KUKA KRL program: EPS_2_251525_MH1778938_A_20251113053654.src

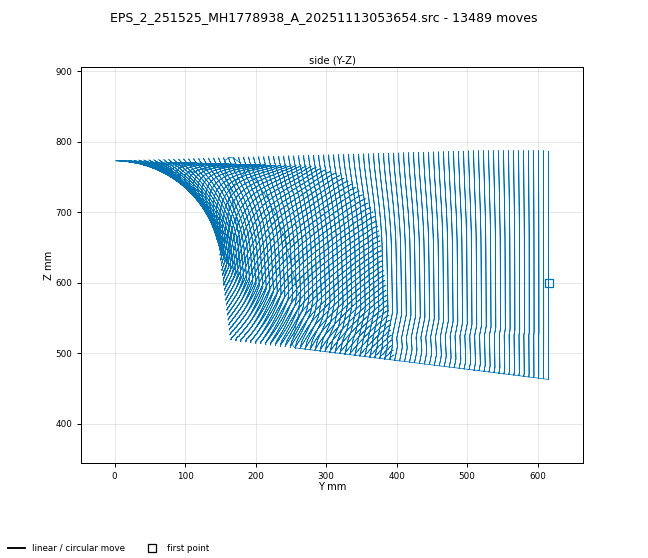
[picture p0: tool path of EPS_2_251525_MH1778938_A_20251113053654.src, 13489 of 13491 moves have a stored position in this frame; points joined in program order, loops and branches not executed]
&ACCESS RVP
&REL 4
&COMMENT QRS 19112012
&PARAM EDITMASK = *
DEF PART()
EXT BAS (BAS_COMMAND :IN,REAL :IN )
INT I
BAS (#INITMOV,0 )

;KUKA QRS Post kuka4.cps  Date:22-06-2017 !

File_ID=2903

QRS_PRE_INIT()

;Init var - Until changes are made in qrs_pre_init
Outlet_Square_prg=0
Inlet_1_Square_prg=0
Inlet_2_Square_prg=0
Inlet_3_Square_prg=0
Inlet_4_Square_prg=0
Inlet_5_Square_prg=0

Outlet_1={X 0.000, Y 516.340, Z 662.000, B 0.000, E1 0.000 }
Inlet_1={X 0.000, Y 535.290, Z 637.000, B 0.000, E1 180.000 }
Outlet_1_type=251
Inlet_1_type=0
;QRS#1=Sidecore dimensions
;QRS#2=250-10" PVC SDR 35
;QRS#3=DeadEnd 251
;QRS#4=
;QRS#5=
;QRS#6=
;QRS#7=
;QRS#8=
;QRS#9=14M PSX
;QRS#10=

;QRS#11=
;QRS#12=
;QRS#13=
;QRS#14=
;QRS#15=
;QRS#16=1220x127x1067 3,5'
;QRS#17=EPS Height
;QRS#18=787,5
;QRS#19=*
;QRS#20= UPDATED VERSION 22-06-2017
;QRS#21=*
Outlet_Square=0100
Inlet_1_Square=00
Inlet_2_Square=0
Inlet_3_Square=0
Inlet_4_Square=0
Inlet_5_Square=0
Mill_Square=1
Outlet_Square_Prg=205
Inlet_1_Square_prg=0

QRS_INIT()

$ADVANCE=5

; T1
PTP {E1 173.595,E2 173.595}
PTP {X 0,Y 615.507,A -85,B 0,C 180,E1 173.595,E2 173.595,E3 0,E4 0,E5 0,E6 0}
QRS_SPEED_INIT()
LIN {X 0,Y 615.507,Z 600,A -85,B 0,C 180,E1 173.595,E2 173.595,E3 0,E4 0,E5 0,E6 0} C_VEL
LIN {X 0,Y 615.507,Z 472.987,A -85,B 0,C 180,E1 173.595,E2 173.595} C_VEL
LIN {X 0,Y 615.507,Z 464.806,A -85,B 0,C 180,E1 173.595,E2 173.595} C_VEL
LIN {X 0,Y 615.49,Z 462.806,A -85,B 0,C 180,E1 173.409,E2 173.409} C_VEL
LIN {X 0,Y 615.478,Z 462.817,A -85,B 0,C 180,E1 170.801,E2 170.801} C_VEL
LIN {X 0,Y 615.479,Z 462.819,A -85,B 0,C 180,E1 168.139,E2 168.139} C_VEL
LIN {X 0,Y 615.488,Z 462.806,A -85,B 0,C 180,E1 165.451,E2 165.451} C_VEL
LIN {X 0,Y 615.479,Z 462.818,A -85,B 0,C 180,E1 162.73,E2 162.73} C_VEL
LIN {X 0,Y 615.477,Z 462.816,A -85,B 0,C 180,E1 159.967,E2 159.967} C_VEL
LIN {X 0,Y 615.482,Z 462.809,A -85,B 0,C 180,E1 157.156,E2 157.156} C_VEL
LIN {X 0,Y 615.494,Z 462.824,A -85,B 0,C 180,E1 154.285,E2 154.285} C_VEL
LIN {X 0,Y 615.486,Z 462.807,A -85,B 0,C 180,E1 151.342,E2 151.342} C_VEL
LIN {X 0,Y 615.477,Z 462.813,A -85,B 0,C 180,E1 148.913,E2 148.913} C_VEL
LIN {X 0,Y 615.485,Z 462.822,A -85,B 0,C 180,E1 146.464,E2 146.464} C_VEL
LIN {X 0,Y 615.481,Z 462.81,A -85,B 0,C 180,E1 143.575,E2 143.575} C_VEL
LIN {X 0,Y 615.479,Z 462.811,A -85,B 0,C 180,E1 140.937,E2 140.937} C_VEL
LIN {X 0,Y 615.482,Z 462.82,A -85,B 0,C 180,E1 138.526,E2 138.526} C_VEL
LIN {X 0,Y 615.478,Z 462.817,A -85,B 0,C 180,E1 135.85,E2 135.85} C_VEL
LIN {X 0,Y 615.485,Z 462.808,A -85,B 0,C 180,E1 133.048,E2 133.048} C_VEL
LIN {X 0,Y 615.49,Z 462.822,A -85,B 0,C 180,E1 130.09,E2 130.09} C_VEL
LIN {X 0,Y 615.49,Z 462.806,A -85,B 0,C 180,E1 127.241,E2 127.241} C_VEL
LIN {X 0,Y 615.476,Z 462.814,A -85,B 0,C 180,E1 124.7,E2 124.7} C_VEL
LIN {X 0,Y 615.488,Z 462.822,A -85,B 0,C 180,E1 122.332,E2 122.332} C_VEL
LIN {X 0,Y 615.478,Z 462.81,A -85,B 0,C 180,E1 119.406,E2 119.406} C_VEL
LIN {X 0,Y 615.491,Z 462.806,A -85,B 0,C 180,E1 117.047,E2 117.047} C_VEL
LIN {X 0,Y 615.487,Z 462.823,A -85,B 0,C 180,E1 114.271,E2 114.271} C_VEL
LIN {X 0,Y 615.48,Z 462.81,A -85,B 0,C 180,E1 111.432,E2 111.432} C_VEL
LIN {X 0,Y 615.477,Z 462.813,A -85,B 0,C 180,E1 108.646,E2 108.646} C_VEL
LIN {X 0,Y 615.486,Z 462.821,A -85,B 0,C 180,E1 105.905,E2 105.905} C_VEL
LIN {X 0,Y 615.487,Z 462.807,A -85,B 0,C 180,E1 103.201,E2 103.201} C_VEL
LIN {X 0,Y 615.476,Z 462.815,A -85,B 0,C 180,E1 100.527,E2 100.527} C_VEL
LIN {X 0,Y 615.487,Z 462.822,A -85,B 0,C 180,E1 97.875,E2 97.875} C_VEL
LIN {X 0,Y 615.479,Z 462.809,A -85,B 0,C 180,E1 95.241,E2 95.241} C_VEL
LIN {X 0,Y 615.478,Z 462.812,A -85,B 0,C 180,E1 92.618,E2 92.618} C_VEL
LIN {X 0,Y 615.486,Z 462.828,A -85,B 0,C 180,E1 90,E2 90} C_VEL
LIN {X 0,Y 615.478,Z 462.812,A -85,B 0,C 180,E1 87.382,E2 87.382} C_VEL
LIN {X 0,Y 615.483,Z 462.808,A -85,B 0,C 180,E1 84.759,E2 84.759} C_VEL
LIN {X 0,Y 615.487,Z 462.822,A -85,B 0,C 180,E1 82.125,E2 82.125} C_VEL
LIN {X 0,Y 615.476,Z 462.815,A -85,B 0,C 180,E1 79.473,E2 79.473} C_VEL
LIN {X 0,Y 615.487,Z 462.807,A -85,B 0,C 180,E1 76.799,E2 76.799} C_VEL
LIN {X 0,Y 615.486,Z 462.821,A -85,B 0,C 180,E1 74.095,E2 74.095} C_VEL
LIN {X 0,Y 615.477,Z 462.813,A -85,B 0,C 180,E1 71.354,E2 71.354} C_VEL
LIN {X 0,Y 615.48,Z 462.81,A -85,B 0,C 180,E1 68.568,E2 68.568} C_VEL
LIN {X 0,Y 615.487,Z 462.823,A -85,B 0,C 180,E1 65.729,E2 65.729} C_VEL
LIN {X 0,Y 615.487,Z 462.807,A -85,B 0,C 180,E1 62.824,E2 62.824} C_VEL
LIN {X 0,Y 615.499,Z 462.825,A -85,B 0,C 180,E1 59.841,E2 59.841} C_VEL
LIN {X 0,Y 615.481,Z 462.819,A -85,B 0,C 180,E1 57.543,E2 57.543} C_VEL
LIN {X 0,Y 615.478,Z 462.812,A -85,B 0,C 180,E1 55.185,E2 55.185} C_VEL
LIN {X 0,Y 615.491,Z 462.806,A -85,B 0,C 180,E1 52.759,E2 52.759} C_VEL
LIN {X 0,Y 615.49,Z 462.822,A -85,B 0,C 180,E1 49.91,E2 49.91} C_VEL
LIN {X 0,Y 615.485,Z 462.808,A -85,B 0,C 180,E1 46.952,E2 46.952} C_VEL
LIN {X 0,Y 615.482,Z 462.82,A -85,B 0,C 180,E1 43.998,E2 43.998} C_VEL
LIN {X 0,Y 615.478,Z 462.811,A -85,B 0,C 180,E1 41.095,E2 41.095} C_VEL
LIN {X 0,Y 615.484,Z 462.808,A -85,B 0,C 180,E1 38.904,E2 38.904} C_VEL
LIN {X 0,Y 615.481,Z 462.81,A -85,B 0,C 180,E1 36.425,E2 36.425} C_VEL
LIN {X 0,Y 615.485,Z 462.822,A -85,B 0,C 180,E1 33.536,E2 33.536} C_VEL
LIN {X 0,Y 615.482,Z 462.809,A -85,B 0,C 180,E1 30.919,E2 30.919} C_VEL
LIN {X 0,Y 615.483,Z 462.808,A -85,B 0,C 180,E1 28.452,E2 28.452} C_VEL
LIN {X 0,Y 615.493,Z 462.824,A -85,B 0,C 180,E1 25.573,E2 25.573} C_VEL
LIN {X 0,Y 615.482,Z 462.809,A -85,B 0,C 180,E1 22.844,E2 22.844} C_VEL
LIN {X 0,Y 615.477,Z 462.816,A -85,B 0,C 180,E1 20.033,E2 20.033} C_VEL
LIN {X 0,Y 615.479,Z 462.818,A -85,B 0,C 180,E1 17.27,E2 17.27} C_VEL
LIN {X 0,Y 615.488,Z 462.806,A -85,B 0,C 180,E1 14.549,E2 14.549} C_VEL
LIN {X 0,Y 615.479,Z 462.819,A -85,B 0,C 180,E1 11.861,E2 11.861} C_VEL
LIN {X 0,Y 615.478,Z 462.817,A -85,B 0,C 180,E1 9.199,E2 9.199} C_VEL
LIN {X 0,Y 615.491,Z 462.806,A -85,B 0,C 180,E1 6.556,E2 6.556} C_VEL
LIN {X 0,Y 615.478,Z 462.817,A -85,B 0,C 180,E1 3.928,E2 3.928} C_VEL
LIN {X 0,Y 615.485,Z 462.821,A -85,B 0,C 180,E1 1.308,E2 1.308} C_VEL
LIN {X 0,Y 615.485,Z 462.808,A -85,B 0,C 180,E1 -1.309,E2 -1.309} C_VEL
LIN {X 0,Y 615.478,Z 462.812,A -85,B 0,C 180,E1 -3.929,E2 -3.929} C_VEL
LIN {X 0,Y 615.489,Z 462.825,A -85,B 0,C 180,E1 -6.591,E2 -6.591} C_VEL
LIN {X 0,Y 615.478,Z 462.811,A -85,B 0,C 180,E1 -9.199,E2 -9.199} C_VEL
LIN {X 0,Y 615.481,Z 462.81,A -85,B 0,C 180,E1 -11.861,E2 -11.861} C_VEL
LIN {X 0,Y 615.488,Z 462.827,A -85,B 0,C 180,E1 -14.549,E2 -14.549} C_VEL
LIN {X 0,Y 615.478,Z 462.811,A -85,B 0,C 180,E1 -17.271,E2 -17.271} C_VEL
LIN {X 0,Y 615.477,Z 462.813,A -85,B 0,C 180,E1 -20.033,E2 -20.033} C_VEL
LIN {X 0,Y 615.482,Z 462.821,A -85,B 0,C 180,E1 -22.845,E2 -22.845} C_VEL
LIN {X 0,Y 615.493,Z 462.805,A -85,B 0,C 180,E1 -25.716,E2 -25.716} C_VEL
LIN {X 0,Y 615.486,Z 462.828,A -85,B 0,C 180,E1 -28.658,E2 -28.658} C_VEL
LIN {X 0,Y 615.477,Z 462.816,A -85,B 0,C 180,E1 -31.087,E2 -31.087} C_VEL
LIN {X 0,Y 615.485,Z 462.808,A -85,B 0,C 180,E1 -33.536,E2 -33.536} C_VEL
LIN {X 0,Y 615.482,Z 462.819,A -85,B 0,C 180,E1 -36.425,E2 -36.425} C_VEL
LIN {X 0,Y 615.478,Z 462.818,A -85,B 0,C 180,E1 -39.063,E2 -39.063} C_VEL
LIN {X 0,Y 615.482,Z 462.809,A -85,B 0,C 180,E1 -41.475,E2 -41.475} C_VEL
LIN {X 0,Y 615.478,Z 462.812,A -85,B 0,C 180,E1 -44.151,E2 -44.151} C_VEL
LIN {X 0,Y 615.485,Z 462.821,A -85,B 0,C 180,E1 -46.953,E2 -46.953} C_VEL
LIN {X 0,Y 615.478,Z 462.812,A -85,B 0,C 180,E1 -49.394,E2 -49.394} C_VEL
LIN {X 0,Y 615.485,Z 462.808,A -85,B 0,C 180,E1 -51.989,E2 -51.989} C_VEL
LIN {X 0,Y 615.474,Z 462.817,A -85,B 0,C 180,E1 -54.384,E2 -54.384} C_VEL
LIN {X 0,Y 615.484,Z 462.827,A -85,B 0,C 180,E1 -56.764,E2 -56.764} C_VEL
LIN {X 0,Y 615.478,Z 462.82,A -85,B 0,C 180,E1 -59.081,E2 -59.081} C_VEL
LIN {X 0,Y 615.48,Z 462.81,A -85,B 0,C 180,E1 -61.551,E2 -61.551} C_VEL
LIN {X 0,Y 615.477,Z 462.813,A -85,B 0,C 180,E1 -64.284,E2 -64.284} C_VEL
LIN {X 0,Y 615.497,Z 463.131,A -85,B 0,C 180,E1 -64.973,E2 -64.973} C_VEL
LIN {X 0,Y 615.483,Z 480.491,A -85,B 0,C 180,E1 -67.655,E2 -67.655} C_VEL
LIN {X 0,Y 615.475,Z 498.123,A -85,B 0,C 180,E1 -70.315,E2 -70.315} C_VEL
LIN {X 0,Y 615.495,Z 516.688,A -85,B 0,C 180,E1 -73.072,E2 -73.072} C_VEL
LIN {X 0,Y 615.49,Z 525.925,A -85,B 0,C 180,E1 -74.393,E2 -74.393} C_VEL
LIN {X 0,Y 615.49,Z 528.646,A -85,B 0,C 180,E1 -74.456,E2 -74.456} C_VEL
LIN {X 0,Y 615.499,Z 662.918,A -85,B 0,C 180,E1 -76.064,E2 -76.064} C_VEL
LIN {X 0,Y 615.497,Z 677.388,A -85,B 0,C 180,E1 -76.379,E2 -76.379} C_VEL
LIN {X 0,Y 615.498,Z 690.696,A -85,B 0,C 180,E1 -76.799,E2 -76.799} C_VEL
LIN {X 0,Y 615.495,Z 702.843,A -85,B 0,C 180,E1 -77.303,E2 -77.303} C_VEL
LIN {X 0,Y 615.492,Z 715.604,A -85,B 0,C 180,E1 -77.972,E2 -77.972} C_VEL
LIN {X 0,Y 615.499,Z 728.344,A -85,B 0,C 180,E1 -78.807,E2 -78.807} C_VEL
LIN {X 0,Y 615.498,Z 738.751,A -85,B 0,C 180,E1 -79.64,E2 -79.64} C_VEL
LIN {X 0,Y 615.497,Z 749.09,A -85,B 0,C 180,E1 -80.636,E2 -80.636} C_VEL
LIN {X 0,Y 615.497,Z 757.604,A -85,B 0,C 180,E1 -81.629,E2 -81.629} C_VEL
LIN {X 0,Y 615.496,Z 765.727,A -85,B 0,C 180,E1 -82.785,E2 -82.785} C_VEL
LIN {X 0,Y 615.497,Z 771.431,A -85,B 0,C 180,E1 -83.773,E2 -83.773} C_VEL
LIN {X 0,Y 615.495,Z 776.081,A -85,B 0,C 180,E1 -84.759,E2 -84.759} C_VEL
LIN {X 0,Y 615.494,Z 780.902,A -85,B 0,C 180,E1 -86.072,E2 -86.072} C_VEL
LIN {X 0,Y 615.496,Z 784.252,A -85,B 0,C 180,E1 -87.382,E2 -87.382} C_VEL
LIN {X 0,Y 615.489,Z 786.229,A -85,B 0,C 180,E1 -88.691,E2 -88.691} C_VEL
LIN {X 0,Y 615.493,Z 786.889,A -85,B 0,C 180,E1 -90,E2 -90} C_VEL
LIN {X 0,Y 615.489,Z 786.229,A -85,B 0,C 180,E1 -91.309,E2 -91.309} C_VEL
LIN {X 0,Y 615.496,Z 784.252,A -85,B 0,C 180,E1 -92.618,E2 -92.618} C_VEL
LIN {X 0,Y 615.494,Z 780.902,A -85,B 0,C 180,E1 -93.928,E2 -93.928} C_VEL
LIN {X 0,Y 615.495,Z 776.081,A -85,B 0,C 180,E1 -95.241,E2 -95.241} C_VEL
LIN {X 0,Y 615.495,Z 769.629,A -85,B 0,C 180,E1 -96.556,E2 -96.556} C_VEL
LIN {X 0,Y 615.497,Z 762.442,A -85,B 0,C 180,E1 -97.71,E2 -97.71} C_VEL
LIN {X 0,Y 615.497,Z 754.905,A -85,B 0,C 180,E1 -98.702,E2 -98.702} C_VEL
LIN {X 0,Y 615.495,Z 745.855,A -85,B 0,C 180,E1 -99.696,E2 -99.696} C_VEL
LIN {X 0,Y 615.497,Z 735.759,A -85,B 0,C 180,E1 -100.618,E2 -100.618} C_VEL
LIN {X 0,Y 615.498,Z 724.861,A -85,B 0,C 180,E1 -101.443,E2 -101.443} C_VEL
LIN {X 0,Y 615.487,Z 712.711,A -85,B 0,C 180,E1 -102.195,E2 -102.195} C_VEL
LIN {X 0,Y 615.494,Z 699.097,A -85,B 0,C 180,E1 -102.865,E2 -102.865} C_VEL
LIN {X 0,Y 615.497,Z 685.843,A -85,B 0,C 180,E1 -103.369,E2 -103.369} C_VEL
LIN {X 0,Y 615.498,Z 672.298,A -85,B 0,C 180,E1 -103.747,E2 -103.747} C_VEL
LIN {X 0,Y 615.497,Z 657.754,A -85,B 0,C 180,E1 -104.013,E2 -104.013} C_VEL
LIN {X 0,Y 615.49,Z 526.279,A -85,B 0,C 180,E1 -105.586,E2 -105.586} C_VEL
LIN {X 0,Y 615.49,Z 524.805,A -85,B 0,C 180,E1 -105.735,E2 -105.735} C_VEL
LIN {X 0,Y 615.479,Z 506.472,A -85,B 0,C 180,E1 -108.44,E2 -108.44} C_VEL
LIN {X 0,Y 615.497,Z 487.671,A -85,B 0,C 180,E1 -111.255,E2 -111.255} C_VEL
LIN {X 0,Y 615.497,Z 469.607,A -85,B 0,C 180,E1 -114.01,E2 -114.01} C_VEL
LIN {X 0,Y 615.497,Z 463,A -85,B 0,C 180,E1 -115.062,E2 -115.062} C_VEL
LIN {X 0,Y 615.487,Z 462.828,A -85,B 0,C 180,E1 -117.177,E2 -117.177} C_VEL
LIN {X 0,Y 615.499,Z 462.804,A -85,B 0,C 180,E1 -120.159,E2 -120.159} C_VEL
LIN {X 0,Y 615.481,Z 462.81,A -85,B 0,C 180,E1 -122.457,E2 -122.457} C_VEL
LIN {X 0,Y 615.477,Z 462.817,A -85,B 0,C 180,E1 -124.815,E2 -124.815} C_VEL
LIN {X 0,Y 615.491,Z 462.826,A -85,B 0,C 180,E1 -127.241,E2 -127.241} C_VEL
LIN {X 0,Y 615.489,Z 462.807,A -85,B 0,C 180,E1 -130.089,E2 -130.089} C_VEL
LIN {X 0,Y 615.49,Z 462.806,A -85,B 0,C 180,E1 -132.352,E2 -132.352} C_VEL
LIN {X 0,Y 615.479,Z 462.822,A -85,B 0,C 180,E1 -135.068,E2 -135.068} C_VEL
LIN {X 0,Y 615.477,Z 462.812,A -85,B 0,C 180,E1 -137.919,E2 -137.919} C_VEL
LIN {X 0,Y 615.498,Z 462.804,A -85,B 0,C 180,E1 -140.25,E2 -140.25} C_VEL
LIN {X 0,Y 615.478,Z 462.821,A -85,B 0,C 180,E1 -143.063,E2 -143.063} C_VEL
LIN {X 0,Y 615.49,Z 462.827,A -85,B 0,C 180,E1 -145.297,E2 -145.297} C_VEL
LIN {X 0,Y 615.479,Z 462.818,A -85,B 0,C 180,E1 -147.668,E2 -147.668} C_VEL
LIN {X 0,Y 615.488,Z 462.807,A -85,B 0,C 180,E1 -150.203,E2 -150.203} C_VEL
LIN {X 0,Y 615.477,Z 462.817,A -85,B 0,C 180,E1 -152.954,E2 -152.954} C_VEL
LIN {X 0,Y 615.479,Z 462.818,A -85,B 0,C 180,E1 -155.727,E2 -155.727} C_VEL
LIN {X 0,Y 615.486,Z 462.808,A -85,B 0,C 180,E1 -158.568,E2 -158.568} C_VEL
LIN {X 0,Y 615.492,Z 462.826,A -85,B 0,C 180,E1 -161.39,E2 -161.39} C_VEL
LIN {X 0,Y 615.48,Z 462.811,A -85,B 0,C 180,E1 -164.094,E2 -164.094} C_VEL
LIN {X 0,Y 615.478,Z 462.812,A -85,B 0,C 180,E1 -166.798,E2 -166.798} C_VEL
LIN {X 0,Y 615.489,Z 462.827,A -85,B 0,C 180,E1 -169.473,E2 -169.473} C_VEL
LIN {X 0,Y 615.479,Z 462.811,A -85,B 0,C 180,E1 -172.124,E2 -172.124} C_VEL
LIN {X 0,Y 615.481,Z 462.81,A -85,B 0,C 180,E1 -174.758,E2 -174.758} C_VEL
LIN {X 0,Y 615.491,Z 462.823,A -85,B 0,C 180,E1 -177.382,E2 -177.382} C_VEL
LIN {X 0,Y 615.477,Z 462.815,A -85,B 0,C 180,E1 -180,E2 -180} C_VEL
LIN {X 0,Y 615.491,Z 462.806,A -85,B 0,C 180,E1 -182.618,E2 -182.618} C_VEL
LIN {X 0,Y 615.476,Z 462.82,A -85,B 0,C 180,E1 -185.241,E2 -185.241} C_VEL
LIN {X 0,Y 615.49,Z 462.806,A -85,B 0,C 180,E1 -186.591,E2 -186.591} C_VEL
LIN {X 0,Y 614.807,Z 462.965,A -85,B 0,C 180,E1 -187.137,E2 -187.137} C_VEL
LIN {X 0,Y 611.966,Z 463.377,A -85,B 0,C 180,E1 -188.023,E2 -188.023} C_VEL
LIN {X 0,Y 609.574,Z 463.69,A -85,B 0,C 180,E1 -188.736,E2 -188.736} C_VEL
LIN {X 0,Y 608.539,Z 463.808,A -85,B 0,C 180,E1 -189.286,E2 -189.286} C_VEL
LIN {X 0,Y 608.451,Z 463.817,A -85,B 0,C 180,E1 -189.472,E2 -189.472} C_VEL
LIN {X 0,Y 608.456,Z 463.815,A -85,B 0,C 180,E1 -192,E2 -192} C_VEL
LIN {X 0,Y 608.472,Z 463.81,A -85,B 0,C 180,E1 -194.72,E2 -194.72} C_VEL
LIN {X 0,Y 608.445,Z 463.821,A -85,B 0,C 180,E1 -197.476,E2 -197.476} C_VEL
LIN {X 0,Y 608.458,Z 463.813,A -85,B 0,C 180,E1 -200.274,E2 -200.274} C_VEL
LIN {X 0,Y 608.449,Z 463.812,A -85,B 0,C 180,E1 -202.477,E2 -202.477} C_VEL
LIN {X 0,Y 608.45,Z 463.817,A -85,B 0,C 180,E1 -205.301,E2 -205.301} C_VEL
LIN {X 0,Y 608.442,Z 463.822,A -85,B 0,C 180,E1 -207.518,E2 -207.518} C_VEL
LIN {X 0,Y 608.464,Z 463.816,A -85,B 0,C 180,E1 -209.973,E2 -209.973} C_VEL
LIN {X 0,Y 608.457,Z 463.812,A -85,B 0,C 180,E1 -212.524,E2 -212.524} C_VEL
LIN {X 0,Y 608.449,Z 463.816,A -85,B 0,C 180,E1 -215.277,E2 -215.277} C_VEL
LIN {X 0,Y 608.46,Z 463.814,A -85,B 0,C 180,E1 -218.241,E2 -218.241} C_VEL
LIN {X 0,Y 608.446,Z 463.814,A -85,B 0,C 180,E1 -220.33,E2 -220.33} C_VEL
LIN {X 0,Y 608.446,Z 463.813,A -85,B 0,C 180,E1 -222.96,E2 -222.96} C_VEL
LIN {X 0,Y 608.459,Z 463.822,A -85,B 0,C 180,E1 -225.735,E2 -225.735} C_VEL
LIN {X 0,Y 608.459,Z 463.811,A -85,B 0,C 180,E1 -228.657,E2 -228.657} C_VEL
LIN {X 0,Y 608.465,Z 463.815,A -85,B 0,C 180,E1 -231.413,E2 -231.413} C_VEL
LIN {X 0,Y 608.47,Z 463.818,A -85,B 0,C 180,E1 -233.951,E2 -233.951} C_VEL
LIN {X 0,Y 608.459,Z 463.814,A -85,B 0,C 180,E1 -236.33,E2 -236.33} C_VEL
LIN {X 0,Y 608.473,Z 463.81,A -85,B 0,C 180,E1 -238.727,E2 -238.727} C_VEL
LIN {X 0,Y 608.466,Z 463.814,A -85,B 0,C 180,E1 -241.38,E2 -241.38} C_VEL
LIN {X 0,Y 608.439,Z 463.823,A -85,B 0,C 180,E1 -243.965,E2 -243.965} C_VEL
LIN {X 0,Y 608.466,Z 463.816,A -85,B 0,C 180,E1 -246.156,E2 -246.156} C_VEL
LIN {X 0,Y 608.467,Z 463.814,A -85,B 0,C 180,E1 -248.309,E2 -248.309} C_VEL
LIN {X 0,Y 608.45,Z 463.813,A -85,B 0,C 180,E1 -251.131,E2 -251.131} C_VEL
LIN {X 0,Y 608.458,Z 463.823,A -85,B 0,C 180,E1 -253.907,E2 -253.907} C_VEL
LIN {X 0,Y 608.464,Z 463.811,A -85,B 0,C 180,E1 -256.644,E2 -256.644} C_VEL
LIN {X 0,Y 608.458,Z 463.813,A -85,B 0,C 180,E1 -259.35,E2 -259.35} C_VEL
LIN {X 0,Y 608.476,Z 463.819,A -85,B 0,C 180,E1 -262.033,E2 -262.033} C_VEL
LIN {X 0,Y 608.46,Z 463.812,A -85,B 0,C 180,E1 -264.698,E2 -264.698} C_VEL
LIN {X 0,Y 608.469,Z 463.811,A -85,B 0,C 180,E1 -267.352,E2 -267.352} C_VEL
LIN {X 0,Y 608.476,Z 463.82,A -85,B 0,C 180,E1 -270,E2 -270} C_VEL
LIN {X 0,Y 608.469,Z 463.811,A -85,B 0,C 180,E1 -272.648,E2 -272.648} C_VEL
LIN {X 0,Y 608.463,Z 463.812,A -85,B 0,C 180,E1 -275.302,E2 -275.302} C_VEL
LIN {X 0,Y 608.476,Z 463.819,A -85,B 0,C 180,E1 -277.967,E2 -277.967} C_VEL
LIN {X 0,Y 608.458,Z 463.813,A -85,B 0,C 180,E1 -280.65,E2 -280.65} C_VEL
LIN {X 0,Y 608.464,Z 463.811,A -85,B 0,C 180,E1 -283.356,E2 -283.356} C_VEL
LIN {X 0,Y 608.458,Z 463.823,A -85,B 0,C 180,E1 -286.093,E2 -286.093} C_VEL
LIN {X 0,Y 608.45,Z 463.813,A -85,B 0,C 180,E1 -288.869,E2 -288.869} C_VEL
LIN {X 0,Y 608.467,Z 463.814,A -85,B 0,C 180,E1 -291.691,E2 -291.691} C_VEL
LIN {X 0,Y 608.454,Z 463.815,A -85,B 0,C 180,E1 -294.57,E2 -294.57} C_VEL
LIN {X 0,Y 608.48,Z 463.809,A -85,B 0,C 180,E1 -297.209,E2 -297.209} C_VEL
LIN {X 0,Y 608.466,Z 463.818,A -85,B 0,C 180,E1 -299.972,E2 -299.972} C_VEL
LIN {X 0,Y 608.456,Z 463.816,A -85,B 0,C 180,E1 -302.522,E2 -302.522} C_VEL
LIN {X 0,Y 608.433,Z 463.814,A -85,B 0,C 180,E1 -305.277,E2 -305.277} C_VEL
LIN {X 0,Y 608.47,Z 463.813,A -85,B 0,C 180,E1 -307.745,E2 -307.745} C_VEL
LIN {X 0,Y 608.474,Z 463.818,A -85,B 0,C 180,E1 -310.332,E2 -310.332} C_VEL
LIN {X 0,Y 608.484,Z 463.807,A -85,B 0,C 180,E1 -313.311,E2 -313.311} C_VEL
LIN {X 0,Y 608.466,Z 463.819,A -85,B 0,C 180,E1 -316.131,E2 -316.131} C_VEL
LIN {X 0,Y 608.448,Z 463.814,A -85,B 0,C 180,E1 -318.823,E2 -318.823} C_VEL
LIN {X 0,Y 608.464,Z 463.811,A -85,B 0,C 180,E1 -321.412,E2 -321.412} C_VEL
LIN {X 0,Y 608.47,Z 463.815,A -85,B 0,C 180,E1 -323.95,E2 -323.95} C_VEL
LIN {X 0,Y 608.461,Z 463.822,A -85,B 0,C 180,E1 -326.33,E2 -326.33} C_VEL
LIN {X 0,Y 608.468,Z 463.814,A -85,B 0,C 180,E1 -328.727,E2 -328.727} C_VEL
LIN {X 0,Y 608.471,Z 463.81,A -85,B 0,C 180,E1 -331.378,E2 -331.378} C_VEL
LIN {X 0,Y 608.475,Z 463.819,A -85,B 0,C 180,E1 -334.276,E2 -334.276} C_VEL
LIN {X 0,Y 608.447,Z 463.815,A -85,B 0,C 180,E1 -336.876,E2 -336.876} C_VEL
LIN {X 0,Y 608.464,Z 463.81,A -85,B 0,C 180,E1 -339.319,E2 -339.319} C_VEL
LIN {X 0,Y 608.446,Z 463.815,A -85,B 0,C 180,E1 -341.828,E2 -341.828} C_VEL
LIN {X 0,Y 608.463,Z 463.818,A -85,B 0,C 180,E1 -344.594,E2 -344.594} C_VEL
LIN {X 0,Y 608.475,Z 463.809,A -85,B 0,C 180,E1 -347.323,E2 -347.323} C_VEL
LIN {X 0,Y 608.45,Z 463.816,A -85,B 0,C 180,E1 -350.023,E2 -350.023} C_VEL
LIN {X 0,Y 608.474,Z 463.816,A -85,B 0,C 180,E1 -352.701,E2 -352.701} C_VEL
LIN {X 0,Y 608.463,Z 463.811,A -85,B 0,C 180,E1 -355.363,E2 -355.363} C_VEL
LIN {X 0,Y 608.448,Z 463.815,A -85,B 0,C 180,E1 -358.015,E2 -358.015} C_VEL
LIN {X 0,Y 608.478,Z 463.817,A -85,B 0,C 180,E1 -360.662,E2 -360.662} C_VEL
LIN {X 0,Y 608.475,Z 463.809,A -85,B 0,C 180,E1 -363.311,E2 -363.311} C_VEL
LIN {X 0,Y 608.453,Z 463.814,A -85,B 0,C 180,E1 -365.967,E2 -365.967} C_VEL
LIN {X 0,Y 608.456,Z 463.821,A -85,B 0,C 180,E1 -368.636,E2 -368.636} C_VEL
LIN {X 0,Y 608.468,Z 463.81,A -85,B 0,C 180,E1 -371.324,E2 -371.324} C_VEL
LIN {X 0,Y 608.458,Z 463.813,A -85,B 0,C 180,E1 -374.038,E2 -374.038} C_VEL
LIN {X 0,Y 608.472,Z 463.817,A -85,B 0,C 180,E1 -376.784,E2 -376.784} C_VEL
LIN {X 0,Y 608.445,Z 463.813,A -85,B 0,C 180,E1 -379.571,E2 -379.571} C_VEL
LIN {X 0,Y 608.467,Z 463.817,A -85,B 0,C 180,E1 -382.406,E2 -382.406} C_VEL
LIN {X 0,Y 608.446,Z 463.823,A -85,B 0,C 180,E1 -384.572,E2 -384.572} C_VEL
LIN {X 0,Y 608.47,Z 463.812,A -85,B 0,C 180,E1 -387.208,E2 -387.208} C_VEL
LIN {X 0,Y 608.464,Z 463.812,A -85,B 0,C 180,E1 -389.973,E2 -389.973} C_VEL
LIN {X 0,Y 608.458,Z 463.82,A -85,B 0,C 180,E1 -392.524,E2 -392.524} C_VEL
LIN {X 0,Y 608.449,Z 463.814,A -85,B 0,C 180,E1 -395.278,E2 -395.278} C_VEL
LIN {X 0,Y 608.461,Z 463.814,A -85,B 0,C 180,E1 -398.241,E2 -398.241} C_VEL
LIN {X 0,Y 608.446,Z 463.817,A -85,B 0,C 180,E1 -400.33,E2 -400.33} C_VEL
LIN {X 0,Y 608.445,Z 463.82,A -85,B 0,C 180,E1 -402.961,E2 -402.961} C_VEL
LIN {X 0,Y 608.459,Z 463.811,A -85,B 0,C 180,E1 -405.736,E2 -405.736} C_VEL
LIN {X 0,Y 608.46,Z 463.82,A -85,B 0,C 180,E1 -408.658,E2 -408.658} C_VEL
LIN {X 0,Y 608.465,Z 463.811,A -85,B 0,C 180,E1 -411.413,E2 -411.413} C_VEL
LIN {X 0,Y 608.443,Z 463.812,A -85,B 0,C 180,E1 -413.955,E2 -413.955} C_VEL
LIN {X 0,Y 608.463,Z 463.814,A -85,B 0,C 180,E1 -416.33,E2 -416.33} C_VEL
LIN {X 0,Y 608.476,Z 463.819,A -85,B 0,C 180,E1 -418.728,E2 -418.728} C_VEL
LIN {X 0,Y 608.466,Z 463.812,A -85,B 0,C 180,E1 -421.382,E2 -421.382} C_VEL
LIN {X 0,Y 608.438,Z 463.815,A -85,B 0,C 180,E1 -423.965,E2 -423.965} C_VEL
LIN {X 0,Y 608.476,Z 463.973,A -85,B 0,C 180,E1 -424.792,E2 -424.792} C_VEL
LIN {X 0,Y 608.561,Z 474.89,A -85,B 0,C 180,E1 -426.521,E2 -426.521} C_VEL
LIN {X 0,Y 608.547,Z 491.17,A -85,B 0,C 180,E1 -429.022,E2 -429.022} C_VEL
LIN {X 0,Y 608.526,Z 510.939,A -85,B 0,C 180,E1 -432.005,E2 -432.005} C_VEL
LIN {X 0,Y 608.506,Z 525.923,A -85,B 0,C 180,E1 -434.209,E2 -434.209} C_VEL
LIN {X 0,Y 608.663,Z 528.646,A -85,B 0,C 180,E1 -434.278,E2 -434.278} C_VEL
LIN {X 0,Y 608.614,Z 663.012,A -85,B 0,C 180,E1 -435.904,E2 -435.904} C_VEL
LIN {X 0,Y 608.599,Z 677.404,A -85,B 0,C 180,E1 -436.222,E2 -436.222} C_VEL
LIN {X 0,Y 608.586,Z 691.839,A -85,B 0,C 180,E1 -436.689,E2 -436.689} C_VEL
LIN {X 0,Y 608.543,Z 704.626,A -85,B 0,C 180,E1 -437.24,E2 -437.24} C_VEL
LIN {X 0,Y 608.531,Z 717.095,A -85,B 0,C 180,E1 -437.917,E2 -437.917} C_VEL
LIN {X 0,Y 608.499,Z 728.475,A -85,B 0,C 180,E1 -438.677,E2 -438.677} C_VEL
LIN {X 0,Y 608.496,Z 738.935,A -85,B 0,C 180,E1 -439.519,E2 -439.519} C_VEL
LIN {X 0,Y 608.479,Z 749.335,A -85,B 0,C 180,E1 -440.527,E2 -440.527} C_VEL
LIN {X 0,Y 608.464,Z 757.911,A -85,B 0,C 180,E1 -441.532,E2 -441.532} C_VEL
LIN {X 0,Y 608.461,Z 766.115,A -85,B 0,C 180,E1 -442.701,E2 -442.701} C_VEL
LIN {X 0,Y 608.443,Z 772.546,A -85,B 0,C 180,E1 -443.831,E2 -443.831} C_VEL
LIN {X 0,Y 608.437,Z 777.961,A -85,B 0,C 180,E1 -445.03,E2 -445.03} C_VEL
LIN {X 0,Y 608.431,Z 781.442,A -85,B 0,C 180,E1 -446.026,E2 -446.026} C_VEL
LIN {X 0,Y 608.424,Z 784.831,A -85,B 0,C 180,E1 -447.352,E2 -447.352} C_VEL
LIN {X 0,Y 608.442,Z 786.83,A -85,B 0,C 180,E1 -448.676,E2 -448.676} C_VEL
LIN {X 0,Y 608.433,Z 787.5,A -85,B 0,C 180,E1 -450,E2 -450} C_VEL
LIN {X 0,Y 608.442,Z 786.83,A -85,B 0,C 180,E1 -451.324,E2 -451.324} C_VEL
LIN {X 0,Y 608.424,Z 784.831,A -85,B 0,C 180,E1 -452.648,E2 -452.648} C_VEL
LIN {X 0,Y 608.431,Z 781.442,A -85,B 0,C 180,E1 -453.974,E2 -453.974} C_VEL
LIN {X 0,Y 608.44,Z 776.569,A -85,B 0,C 180,E1 -455.302,E2 -455.302} C_VEL
LIN {X 0,Y 608.445,Z 770.212,A -85,B 0,C 180,E1 -456.603,E2 -456.603} C_VEL
LIN {X 0,Y 608.453,Z 762.797,A -85,B 0,C 180,E1 -457.8,E2 -457.8} C_VEL
LIN {X 0,Y 608.473,Z 753.825,A -85,B 0,C 180,E1 -458.97,E2 -458.97} C_VEL
LIN {X 0,Y 608.472,Z 744.391,A -85,B 0,C 180,E1 -459.977,E2 -459.977} C_VEL
LIN {X 0,Y 608.506,Z 733.043,A -85,B 0,C 180,E1 -460.973,E2 -460.973} C_VEL
LIN {X 0,Y 608.532,Z 721.15,A -85,B 0,C 180,E1 -461.829,E2 -461.829} C_VEL
LIN {X 0,Y 608.529,Z 708.082,A -85,B 0,C 180,E1 -462.591,E2 -462.591} C_VEL
LIN {X 0,Y 608.563,Z 695.165,A -85,B 0,C 180,E1 -463.184,E2 -463.184} C_VEL
LIN {X 0,Y 608.601,Z 681.926,A -85,B 0,C 180,E1 -463.651,E2 -463.651} C_VEL
LIN {X 0,Y 608.621,Z 667.482,A -85,B 0,C 180,E1 -464.012,E2 -464.012} C_VEL
LIN {X 0,Y 608.627,Z 651.188,A -85,B 0,C 180,E1 -464.257,E2 -464.257} C_VEL
LIN {X 0,Y 608.587,Z 526.547,A -85,B 0,C 180,E1 -465.757,E2 -465.757} C_VEL
LIN {X 0,Y 608.515,Z 525.52,A -85,B 0,C 180,E1 -465.834,E2 -465.834} C_VEL
LIN {X 0,Y 608.495,Z 507.601,A -85,B 0,C 180,E1 -468.496,E2 -468.496} C_VEL
LIN {X 0,Y 608.553,Z 488.845,A -85,B 0,C 180,E1 -471.332,E2 -471.332} C_VEL
LIN {X 0,Y 608.598,Z 470.389,A -85,B 0,C 180,E1 -474.177,E2 -474.177} C_VEL
LIN {X 0,Y 608.469,Z 463.915,A -85,B 0,C 180,E1 -475.231,E2 -475.231} C_VEL
LIN {X 0,Y 608.449,Z 463.817,A -85,B 0,C 180,E1 -477.517,E2 -477.517} C_VEL
LIN {X 0,Y 608.466,Z 463.811,A -85,B 0,C 180,E1 -479.971,E2 -479.971} C_VEL
LIN {X 0,Y 608.457,Z 463.813,A -85,B 0,C 180,E1 -482.521,E2 -482.521} C_VEL
LIN {X 0,Y 608.433,Z 463.823,A -85,B 0,C 180,E1 -485.277,E2 -485.277} C_VEL
LIN {X 0,Y 608.47,Z 463.812,A -85,B 0,C 180,E1 -487.745,E2 -487.745} C_VEL
LIN {X 0,Y 608.45,Z 463.812,A -85,B 0,C 180,E1 -490.329,E2 -490.329} C_VEL
LIN {X 0,Y 608.484,Z 463.818,A -85,B 0,C 180,E1 -493.31,E2 -493.31} C_VEL
LIN {X 0,Y 608.466,Z 463.81,A -85,B 0,C 180,E1 -496.13,E2 -496.13} C_VEL
LIN {X 0,Y 608.448,Z 463.816,A -85,B 0,C 180,E1 -498.823,E2 -498.823} C_VEL
LIN {X 0,Y 608.462,Z 463.82,A -85,B 0,C 180,E1 -501.411,E2 -501.411} C_VEL
LIN {X 0,Y 608.473,Z 463.811,A -85,B 0,C 180,E1 -503.949,E2 -503.949} C_VEL
LIN {X 0,Y 608.461,Z 463.811,A -85,B 0,C 180,E1 -506.329,E2 -506.329} C_VEL
LIN {X 0,Y 608.47,Z 463.811,A -85,B 0,C 180,E1 -508.727,E2 -508.727} C_VEL
LIN {X 0,Y 608.471,Z 463.82,A -85,B 0,C 180,E1 -511.378,E2 -511.378} C_VEL
LIN {X 0,Y 608.475,Z 463.809,A -85,B 0,C 180,E1 -514.276,E2 -514.276} C_VEL
LIN {X 0,Y 608.447,Z 463.815,A -85,B 0,C 180,E1 -516.876,E2 -516.876} C_VEL
LIN {X 0,Y 608.465,Z 463.82,A -85,B 0,C 180,E1 -519.319,E2 -519.319} C_VEL
LIN {X 0,Y 608.446,Z 463.817,A -85,B 0,C 180,E1 -521.828,E2 -521.828} C_VEL
LIN {X 0,Y 608.463,Z 463.811,A -85,B 0,C 180,E1 -524.594,E2 -524.594} C_VEL
LIN {X 0,Y 608.474,Z 463.818,A -85,B 0,C 180,E1 -527.323,E2 -527.323} C_VEL
LIN {X 0,Y 608.45,Z 463.814,A -85,B 0,C 180,E1 -530.022,E2 -530.022} C_VEL
LIN {X 0,Y 608.455,Z 463.812,A -85,B 0,C 180,E1 -532.7,E2 -532.7} C_VEL
LIN {X 0,Y 608.461,Z 463.819,A -85,B 0,C 180,E1 -535.362,E2 -535.362} C_VEL
LIN {X 0,Y 608.448,Z 463.815,A -85,B 0,C 180,E1 -538.014,E2 -538.014} C_VEL
LIN {X 0,Y 608.478,Z 463.809,A -85,B 0,C 180,E1 -540.661,E2 -540.661} C_VEL
LIN {X 0,Y 608.474,Z 463.816,A -85,B 0,C 180,E1 -543.31,E2 -543.31} C_VEL
LIN {X 0,Y 608.453,Z 463.816,A -85,B 0,C 180,E1 -545.967,E2 -545.967} C_VEL
LIN {X 0,Y 608.456,Z 463.811,A -85,B 0,C 180,E1 -548.636,E2 -548.636} C_VEL
LIN {X 0,Y 608.451,Z 463.817,A -85,B 0,C 180,E1 -549.472,E2 -549.472} C_VEL
LIN {X 0,Y 607.773,Z 463.9,A -85,B 0,C 180,E1 -550.024,E2 -550.024} C_VEL
LIN {X 0,Y 604.919,Z 464.254,A -85,B 0,C 180,E1 -550.921,E2 -550.921} C_VEL
LIN {X 0,Y 602.516,Z 464.561,A -85,B 0,C 180,E1 -551.643,E2 -551.643} C_VEL
LIN {X 0,Y 601.488,Z 464.682,A -85,B 0,C 180,E1 -552.2,E2 -552.2} C_VEL
LIN {X 0,Y 601.405,Z 464.69,A -85,B 0,C 180,E1 -552.388,E2 -552.388} C_VEL
LIN {X 0,Y 601.425,Z 464.688,A -85,B 0,C 180,E1 -554.897,E2 -554.897} C_VEL
LIN {X 0,Y 601.426,Z 464.688,A -85,B 0,C 180,E1 -556.986,E2 -556.986} C_VEL
LIN {X 0,Y 601.4,Z 464.698,A -85,B 0,C 180,E1 -559.809,E2 -559.809} C_VEL
LIN {X 0,Y 601.405,Z 464.69,A -85,B 0,C 180,E1 -562.606,E2 -562.606} C_VEL
LIN {X 0,Y 601.397,Z 464.691,A -85,B 0,C 180,E1 -564.878,E2 -564.878} C_VEL
LIN {X 0,Y 601.415,Z 464.696,A -85,B 0,C 180,E1 -567.867,E2 -567.867} C_VEL
LIN {X 0,Y 601.438,Z 464.688,A -85,B 0,C 180,E1 -570.163,E2 -570.163} C_VEL
LIN {X 0,Y 601.416,Z 464.688,A -85,B 0,C 180,E1 -572.717,E2 -572.717} C_VEL
LIN {X 0,Y 601.414,Z 464.691,A -85,B 0,C 180,E1 -575.116,E2 -575.116} C_VEL
LIN {X 0,Y 601.425,Z 464.693,A -85,B 0,C 180,E1 -577.419,E2 -577.419} C_VEL
LIN {X 0,Y 601.406,Z 464.695,A -85,B 0,C 180,E1 -579.995,E2 -579.995} C_VEL
LIN {X 0,Y 601.403,Z 464.69,A -85,B 0,C 180,E1 -582.67,E2 -582.67} C_VEL
LIN {X 0,Y 601.417,Z 464.694,A -85,B 0,C 180,E1 -585.482,E2 -585.482} C_VEL
LIN {X 0,Y 601.421,Z 464.689,A -85,B 0,C 180,E1 -588.406,E2 -588.406} C_VEL
LIN {X 0,Y 601.431,Z 464.687,A -85,B 0,C 180,E1 -590.876,E2 -590.876} C_VEL
LIN {X 0,Y 601.437,Z 464.695,A -85,B 0,C 180,E1 -593.734,E2 -593.734} C_VEL
LIN {X 0,Y 601.422,Z 464.688,A -85,B 0,C 180,E1 -596.687,E2 -596.687} C_VEL
LIN {X 0,Y 601.428,Z 464.688,A -85,B 0,C 180,E1 -599.059,E2 -599.059} C_VEL
LIN {X 0,Y 601.425,Z 464.691,A -85,B 0,C 180,E1 -601.374,E2 -601.374} C_VEL
LIN {X 0,Y 601.399,Z 464.698,A -85,B 0,C 180,E1 -603.637,E2 -603.637} C_VEL
LIN {X 0,Y 601.416,Z 464.69,A -85,B 0,C 180,E1 -606.59,E2 -606.59} C_VEL
LIN {X 0,Y 601.425,Z 464.692,A -85,B 0,C 180,E1 -609.478,E2 -609.478} C_VEL
LIN {X 0,Y 601.396,Z 464.695,A -85,B 0,C 180,E1 -612.312,E2 -612.312} C_VEL
LIN {X 0,Y 601.415,Z 464.692,A -85,B 0,C 180,E1 -614.409,E2 -614.409} C_VEL
LIN {X 0,Y 601.415,Z 464.689,A -85,B 0,C 180,E1 -617.172,E2 -617.172} C_VEL
LIN {X 0,Y 601.43,Z 464.698,A -85,B 0,C 180,E1 -619.905,E2 -619.905} C_VEL
LIN {X 0,Y 601.452,Z 464.686,A -85,B 0,C 180,E1 -622.615,E2 -622.615} C_VEL
LIN {X 0,Y 601.415,Z 464.69,A -85,B 0,C 180,E1 -625.308,E2 -625.308} C_VEL
LIN {X 0,Y 601.433,Z 464.698,A -85,B 0,C 180,E1 -627.991,E2 -627.991} C_VEL
LIN {X 0,Y 601.442,Z 464.687,A -85,B 0,C 180,E1 -630.67,E2 -630.67} C_VEL
LIN {X 0,Y 601.427,Z 464.689,A -85,B 0,C 180,E1 -633.349,E2 -633.349} C_VEL
LIN {X 0,Y 601.411,Z 464.7,A -85,B 0,C 180,E1 -636.037,E2 -636.037} C_VEL
LIN {X 0,Y 601.438,Z 464.697,A -85,B 0,C 180,E1 -638.061,E2 -638.061} C_VEL
LIN {X 0,Y 601.423,Z 464.688,A -85,B 0,C 180,E1 -641.013,E2 -641.013} C_VEL
LIN {X 0,Y 601.417,Z 464.691,A -85,B 0,C 180,E1 -643.516,E2 -643.516} C_VEL
LIN {X 0,Y 601.435,Z 464.694,A -85,B 0,C 180,E1 -646.287,E2 -646.287} C_VEL
LIN {X 0,Y 601.414,Z 464.689,A -85,B 0,C 180,E1 -649.099,E2 -649.099} C_VEL
LIN {X 0,Y 601.414,Z 464.697,A -85,B 0,C 180,E1 -651.959,E2 -651.959} C_VEL
LIN {X 0,Y 601.437,Z 464.694,A -85,B 0,C 180,E1 -654.294,E2 -654.294} C_VEL
LIN {X 0,Y 601.452,Z 464.684,A -85,B 0,C 180,E1 -657.11,E2 -657.11} C_VEL
LIN {X 0,Y 601.443,Z 464.697,A -85,B 0,C 180,E1 -660.162,E2 -660.162} C_VEL
LIN {X 0,Y 601.417,Z 464.691,A -85,B 0,C 180,E1 -662.716,E2 -662.716} C_VEL
LIN {X 0,Y 601.402,Z 464.69,A -85,B 0,C 180,E1 -665.114,E2 -665.114} C_VEL
LIN {X 0,Y 601.431,Z 464.686,A -85,B 0,C 180,E1 -667.418,E2 -667.418} C_VEL
LIN {X 0,Y 601.407,Z 464.697,A -85,B 0,C 180,E1 -669.994,E2 -669.994} C_VEL
LIN {X 0,Y 601.431,Z 464.688,A -85,B 0,C 180,E1 -672.667,E2 -672.667} C_VEL
LIN {X 0,Y 601.416,Z 464.689,A -85,B 0,C 180,E1 -675.482,E2 -675.482} C_VEL
LIN {X 0,Y 601.417,Z 464.696,A -85,B 0,C 180,E1 -678.406,E2 -678.406} C_VEL
LIN {X 0,Y 601.43,Z 464.689,A -85,B 0,C 180,E1 -680.875,E2 -680.875} C_VEL
LIN {X 0,Y 601.435,Z 464.688,A -85,B 0,C 180,E1 -683.733,E2 -683.733} C_VEL
LIN {X 0,Y 601.428,Z 464.693,A -85,B 0,C 180,E1 -686.063,E2 -686.063} C_VEL
LIN {X 0,Y 601.433,Z 464.693,A -85,B 0,C 180,E1 -688.541,E2 -688.541} C_VEL
LIN {X 0,Y 601.43,Z 464.687,A -85,B 0,C 180,E1 -691.374,E2 -691.374} C_VEL
LIN {X 0,Y 601.415,Z 464.695,A -85,B 0,C 180,E1 -694.13,E2 -694.13} C_VEL
LIN {X 0,Y 601.415,Z 464.695,A -85,B 0,C 180,E1 -696.59,E2 -696.59} C_VEL
LIN {X 0,Y 601.427,Z 464.687,A -85,B 0,C 180,E1 -699.478,E2 -699.478} C_VEL
LIN {X 0,Y 601.392,Z 464.701,A -85,B 0,C 180,E1 -702.312,E2 -702.312} C_VEL
LIN {X 0,Y 601.409,Z 464.7,A -85,B 0,C 180,E1 -704.409,E2 -704.409} C_VEL
LIN {X 0,Y 601.418,Z 464.689,A -85,B 0,C 180,E1 -707.172,E2 -707.172} C_VEL
LIN {X 0,Y 601.428,Z 464.689,A -85,B 0,C 180,E1 -709.905,E2 -709.905} C_VEL
LIN {X 0,Y 601.444,Z 464.693,A -85,B 0,C 180,E1 -712.615,E2 -712.615} C_VEL
LIN {X 0,Y 601.429,Z 464.687,A -85,B 0,C 180,E1 -715.308,E2 -715.308} C_VEL
LIN {X 0,Y 601.418,Z 464.69,A -85,B 0,C 180,E1 -717.991,E2 -717.991} C_VEL
LIN {X 0,Y 601.448,Z 464.692,A -85,B 0,C 180,E1 -720.67,E2 -720.67} C_VEL
LIN {X 0,Y 601.426,Z 464.687,A -85,B 0,C 180,E1 -723.35,E2 -723.35} C_VEL
LIN {X 0,Y 601.406,Z 464.692,A -85,B 0,C 180,E1 -726.037,E2 -726.037} C_VEL
LIN {X 0,Y 601.434,Z 464.694,A -85,B 0,C 180,E1 -728.738,E2 -728.738} C_VEL
LIN {X 0,Y 601.427,Z 464.687,A -85,B 0,C 180,E1 -731.459,E2 -731.459} C_VEL
LIN {X 0,Y 601.41,Z 464.693,A -85,B 0,C 180,E1 -734.206,E2 -734.206} C_VEL
LIN {X 0,Y 601.426,Z 464.691,A -85,B 0,C 180,E1 -736.986,E2 -736.986} C_VEL
LIN {X 0,Y 601.4,Z 464.69,A -85,B 0,C 180,E1 -739.81,E2 -739.81} C_VEL
LIN {X 0,Y 601.406,Z 464.7,A -85,B 0,C 180,E1 -742.606,E2 -742.606} C_VEL
LIN {X 0,Y 601.398,Z 464.697,A -85,B 0,C 180,E1 -744.879,E2 -744.879} C_VEL
LIN {X 0,Y 601.416,Z 464.688,A -85,B 0,C 180,E1 -747.868,E2 -747.868} C_VEL
LIN {X 0,Y 601.421,Z 464.691,A -85,B 0,C 180,E1 -750.165,E2 -750.165} C_VEL
LIN {X 0,Y 601.417,Z 464.698,A -85,B 0,C 180,E1 -752.717,E2 -752.717} C_VEL
LIN {X 0,Y 601.414,Z 464.692,A -85,B 0,C 180,E1 -755.116,E2 -755.116} C_VEL
LIN {X 0,Y 601.428,Z 464.688,A -85,B 0,C 180,E1 -757.42,E2 -757.42} C_VEL
LIN {X 0,Y 601.406,Z 464.691,A -85,B 0,C 180,E1 -759.996,E2 -759.996} C_VEL
LIN {X 0,Y 601.405,Z 464.7,A -85,B 0,C 180,E1 -762.671,E2 -762.671} C_VEL
LIN {X 0,Y 601.421,Z 464.688,A -85,B 0,C 180,E1 -765.483,E2 -765.483} C_VEL
LIN {X 0,Y 601.423,Z 464.692,A -85,B 0,C 180,E1 -768.407,E2 -768.407} C_VEL
LIN {X 0,Y 601.432,Z 464.695,A -85,B 0,C 180,E1 -770.876,E2 -770.876} C_VEL
LIN {X 0,Y 601.399,Z 464.69,A -85,B 0,C 180,E1 -773.418,E2 -773.418} C_VEL
LIN {X 0,Y 601.429,Z 464.688,A -85,B 0,C 180,E1 -776.065,E2 -776.065} C_VEL
LIN {X 0,Y 601.44,Z 464.691,A -85,B 0,C 180,E1 -778.543,E2 -778.543} C_VEL
LIN {X 0,Y 601.426,Z 464.69,A -85,B 0,C 180,E1 -781.374,E2 -781.374} C_VEL
LIN {X 0,Y 601.4,Z 464.694,A -85,B 0,C 180,E1 -783.637,E2 -783.637} C_VEL
LIN {X 0,Y 601.465,Z 464.928,A -85,B 0,C 180,E1 -784.64,E2 -784.64} C_VEL
LIN {X 0,Y 601.696,Z 471.188,A -85,B 0,C 180,E1 -785.653,E2 -785.653} C_VEL
LIN {X 0,Y 601.636,Z 488.845,A -85,B 0,C 180,E1 -788.41,E2 -788.41} C_VEL
LIN {X 0,Y 601.521,Z 506.753,A -85,B 0,C 180,E1 -791.153,E2 -791.153} C_VEL
LIN {X 0,Y 601.509,Z 523.731,A -85,B 0,C 180,E1 -793.715,E2 -793.715} C_VEL
LIN {X 0,Y 601.538,Z 526.264,A -85,B 0,C 180,E1 -794.043,E2 -794.043} C_VEL
LIN {X 0,Y 601.839,Z 528.646,A -85,B 0,C 180,E1 -794.095,E2 -794.095} C_VEL
LIN {X 0,Y 601.737,Z 663.017,A -85,B 0,C 180,E1 -795.74,E2 -795.74} C_VEL
LIN {X 0,Y 601.711,Z 677.511,A -85,B 0,C 180,E1 -796.063,E2 -796.063} C_VEL
LIN {X 0,Y 601.668,Z 691.839,A -85,B 0,C 180,E1 -796.533,E2 -796.533} C_VEL
LIN {X 0,Y 601.605,Z 704.616,A -85,B 0,C 180,E1 -797.09,E2 -797.09} C_VEL
LIN {X 0,Y 601.545,Z 717.095,A -85,B 0,C 180,E1 -797.775,E2 -797.775} C_VEL
LIN {X 0,Y 601.504,Z 728.479,A -85,B 0,C 180,E1 -798.543,E2 -798.543} C_VEL
LIN {X 0,Y 601.482,Z 738.939,A -85,B 0,C 180,E1 -799.396,E2 -799.396} C_VEL
LIN {X 0,Y 601.43,Z 749.327,A -85,B 0,C 180,E1 -800.415,E2 -800.415} C_VEL
LIN {X 0,Y 601.407,Z 757.903,A -85,B 0,C 180,E1 -801.431,E2 -801.431} C_VEL
LIN {X 0,Y 601.392,Z 766.118,A -85,B 0,C 180,E1 -802.614,E2 -802.614} C_VEL
LIN {X 0,Y 601.361,Z 771.753,A -85,B 0,C 180,E1 -803.605,E2 -803.605} C_VEL
LIN {X 0,Y 601.355,Z 776.572,A -85,B 0,C 180,E1 -804.635,E2 -804.635} C_VEL
LIN {X 0,Y 601.343,Z 781.444,A -85,B 0,C 180,E1 -805.979,E2 -805.979} C_VEL
LIN {X 0,Y 601.323,Z 784.83,A -85,B 0,C 180,E1 -807.32,E2 -807.32} C_VEL
LIN {X 0,Y 601.342,Z 786.827,A -85,B 0,C 180,E1 -808.661,E2 -808.661} C_VEL
LIN {X 0,Y 601.333,Z 787.5,A -85,B 0,C 180,E1 -810,E2 -810} C_VEL
LIN {X 0,Y 601.342,Z 786.827,A -85,B 0,C 180,E1 -811.339,E2 -811.339} C_VEL
LIN {X 0,Y 601.323,Z 784.83,A -85,B 0,C 180,E1 -812.68,E2 -812.68} C_VEL
LIN {X 0,Y 601.343,Z 781.444,A -85,B 0,C 180,E1 -814.021,E2 -814.021} C_VEL
LIN {X 0,Y 601.355,Z 776.572,A -85,B 0,C 180,E1 -815.365,E2 -815.365} C_VEL
LIN {X 0,Y 601.355,Z 770.053,A -85,B 0,C 180,E1 -816.711,E2 -816.711} C_VEL
LIN {X 0,Y 601.398,Z 762.793,A -85,B 0,C 180,E1 -817.892,E2 -817.892} C_VEL
LIN {X 0,Y 601.43,Z 753.825,A -85,B 0,C 180,E1 -819.076,E2 -819.076} C_VEL
LIN {X 0,Y 601.44,Z 744.389,A -85,B 0,C 180,E1 -820.095,E2 -820.095} C_VEL
LIN {X 0,Y 601.505,Z 733.682,A -85,B 0,C 180,E1 -821.05,E2 -821.05} C_VEL
LIN {X 0,Y 601.543,Z 722.427,A -85,B 0,C 180,E1 -821.883,E2 -821.883} C_VEL
LIN {X 0,Y 601.563,Z 709.654,A -85,B 0,C 180,E1 -822.653,E2 -822.653} C_VEL
LIN {X 0,Y 601.632,Z 696.189,A -85,B 0,C 180,E1 -823.296,E2 -823.296} C_VEL
LIN {X 0,Y 601.701,Z 682.77,A -85,B 0,C 180,E1 -823.783,E2 -823.783} C_VEL
LIN {X 0,Y 601.753,Z 668.563,A -85,B 0,C 180,E1 -824.154,E2 -824.154} C_VEL
LIN {X 0,Y 601.755,Z 653.154,A -85,B 0,C 180,E1 -824.4,E2 -824.4} C_VEL
LIN {X 0,Y 601.777,Z 527.639,A -85,B 0,C 180,E1 -825.919,E2 -825.919} C_VEL
LIN {X 0,Y 601.525,Z 525.918,A -85,B 0,C 180,E1 -825.979,E2 -825.979} C_VEL
LIN {X 0,Y 601.524,Z 509.776,A -85,B 0,C 180,E1 -828.388,E2 -828.388} C_VEL
LIN {X 0,Y 601.611,Z 491.17,A -85,B 0,C 180,E1 -831.231,E2 -831.231} C_VEL
LIN {X 0,Y 601.673,Z 472.564,A -85,B 0,C 180,E1 -834.131,E2 -834.131} C_VEL
LIN {X 0,Y 601.57,Z 465.587,A -85,B 0,C 180,E1 -835.24,E2 -835.24} C_VEL
LIN {X 0,Y 601.435,Z 464.758,A -85,B 0,C 180,E1 -835.431,E2 -835.431} C_VEL
LIN {X 0,Y 601.403,Z 464.691,A -85,B 0,C 180,E1 -837.868,E2 -837.868} C_VEL
LIN {X 0,Y 601.427,Z 464.687,A -85,B 0,C 180,E1 -840.163,E2 -840.163} C_VEL
LIN {X 0,Y 601.419,Z 464.691,A -85,B 0,C 180,E1 -842.715,E2 -842.715} C_VEL
LIN {X 0,Y 601.39,Z 464.701,A -85,B 0,C 180,E1 -845.111,E2 -845.111} C_VEL
LIN {X 0,Y 601.434,Z 464.693,A -85,B 0,C 180,E1 -847.418,E2 -847.418} C_VEL
LIN {X 0,Y 601.408,Z 464.69,A -85,B 0,C 180,E1 -849.994,E2 -849.994} C_VEL
LIN {X 0,Y 601.411,Z 464.691,A -85,B 0,C 180,E1 -852.669,E2 -852.669} C_VEL
LIN {X 0,Y 601.421,Z 464.695,A -85,B 0,C 180,E1 -855.481,E2 -855.481} C_VEL
LIN {X 0,Y 601.418,Z 464.688,A -85,B 0,C 180,E1 -858.406,E2 -858.406} C_VEL
LIN {X 0,Y 601.43,Z 464.691,A -85,B 0,C 180,E1 -860.875,E2 -860.875} C_VEL
LIN {X 0,Y 601.438,Z 464.69,A -85,B 0,C 180,E1 -863.733,E2 -863.733} C_VEL
LIN {X 0,Y 601.429,Z 464.687,A -85,B 0,C 180,E1 -866.063,E2 -866.063} C_VEL
LIN {X 0,Y 601.435,Z 464.686,A -85,B 0,C 180,E1 -868.541,E2 -868.541} C_VEL
LIN {X 0,Y 601.43,Z 464.697,A -85,B 0,C 180,E1 -871.373,E2 -871.373} C_VEL
LIN {X 0,Y 601.416,Z 464.689,A -85,B 0,C 180,E1 -874.129,E2 -874.129} C_VEL
LIN {X 0,Y 601.416,Z 464.689,A -85,B 0,C 180,E1 -876.589,E2 -876.589} C_VEL
LIN {X 0,Y 601.428,Z 464.696,A -85,B 0,C 180,E1 -879.478,E2 -879.478} C_VEL
LIN {X 0,Y 601.391,Z 464.692,A -85,B 0,C 180,E1 -882.311,E2 -882.311} C_VEL
LIN {X 0,Y 601.408,Z 464.689,A -85,B 0,C 180,E1 -884.408,E2 -884.408} C_VEL
LIN {X 0,Y 601.417,Z 464.693,A -85,B 0,C 180,E1 -887.172,E2 -887.172} C_VEL
LIN {X 0,Y 601.428,Z 464.69,A -85,B 0,C 180,E1 -889.905,E2 -889.905} C_VEL
LIN {X 0,Y 601.432,Z 464.686,A -85,B 0,C 180,E1 -892.614,E2 -892.614} C_VEL
LIN {X 0,Y 601.428,Z 464.694,A -85,B 0,C 180,E1 -895.308,E2 -895.308} C_VEL
LIN {X 0,Y 601.418,Z 464.691,A -85,B 0,C 180,E1 -897.991,E2 -897.991} C_VEL
LIN {X 0,Y 601.448,Z 464.684,A -85,B 0,C 180,E1 -900.669,E2 -900.669} C_VEL
LIN {X 0,Y 601.426,Z 464.694,A -85,B 0,C 180,E1 -903.349,E2 -903.349} C_VEL
LIN {X 0,Y 601.406,Z 464.693,A -85,B 0,C 180,E1 -906.037,E2 -906.037} C_VEL
LIN {X 0,Y 601.434,Z 464.686,A -85,B 0,C 180,E1 -908.737,E2 -908.737} C_VEL
LIN {X 0,Y 601.426,Z 464.696,A -85,B 0,C 180,E1 -911.458,E2 -911.458} C_VEL
LIN {X 0,Y 601.405,Z 464.69,A -85,B 0,C 180,E1 -912.388,E2 -912.388} C_VEL
LIN {X 0,Y 600.742,Z 464.774,A -85,B 0,C 180,E1 -912.947,E2 -912.947} C_VEL
LIN {X 0,Y 597.891,Z 465.134,A -85,B 0,C 180,E1 -913.855,E2 -913.855} C_VEL
LIN {X 0,Y 595.479,Z 465.432,A -85,B 0,C 180,E1 -914.585,E2 -914.585} C_VEL
LIN {X 0,Y 594.441,Z 465.561,A -85,B 0,C 180,E1 -915.149,E2 -915.149} C_VEL
LIN {X 0,Y 594.355,Z 465.571,A -85,B 0,C 180,E1 -915.34,E2 -915.34} C_VEL
LIN {X 0,Y 594.373,Z 465.571,A -85,B 0,C 180,E1 -917.904,E2 -917.904} C_VEL
LIN {X 0,Y 594.375,Z 465.567,A -85,B 0,C 180,E1 -920.919,E2 -920.919} C_VEL
LIN {X 0,Y 594.383,Z 465.573,A -85,B 0,C 180,E1 -923.704,E2 -923.704} C_VEL
LIN {X 0,Y 594.378,Z 465.565,A -85,B 0,C 180,E1 -926.699,E2 -926.699} C_VEL
LIN {X 0,Y 594.377,Z 465.566,A -85,B 0,C 180,E1 -928.998,E2 -928.998} C_VEL
LIN {X 0,Y 594.384,Z 465.574,A -85,B 0,C 180,E1 -931.646,E2 -931.646} C_VEL
LIN {X 0,Y 594.392,Z 465.563,A -85,B 0,C 180,E1 -934.579,E2 -934.579} C_VEL
LIN {X 0,Y 594.377,Z 465.567,A -85,B 0,C 180,E1 -937.087,E2 -937.087} C_VEL
LIN {X 0,Y 594.372,Z 465.576,A -85,B 0,C 180,E1 -939.775,E2 -939.775} C_VEL
LIN {X 0,Y 594.361,Z 465.569,A -85,B 0,C 180,E1 -942.375,E2 -942.375} C_VEL
LIN {X 0,Y 594.354,Z 465.57,A -85,B 0,C 180,E1 -945.192,E2 -945.192} C_VEL
LIN {X 0,Y 594.381,Z 465.57,A -85,B 0,C 180,E1 -947.627,E2 -947.627} C_VEL
LIN {X 0,Y 594.386,Z 465.567,A -85,B 0,C 180,E1 -950.321,E2 -950.321} C_VEL
LIN {X 0,Y 594.381,Z 465.564,A -85,B 0,C 180,E1 -952.914,E2 -952.914} C_VEL
LIN {X 0,Y 594.377,Z 465.576,A -85,B 0,C 180,E1 -955.861,E2 -955.861} C_VEL
LIN {X 0,Y 594.386,Z 465.565,A -85,B 0,C 180,E1 -958.651,E2 -958.651} C_VEL
LIN {X 0,Y 594.377,Z 465.566,A -85,B 0,C 180,E1 -961.042,E2 -961.042} C_VEL
LIN {X 0,Y 594.38,Z 465.574,A -85,B 0,C 180,E1 -963.977,E2 -963.977} C_VEL
LIN {X 0,Y 594.388,Z 465.568,A -85,B 0,C 180,E1 -966.297,E2 -966.297} C_VEL
LIN {X 0,Y 594.397,Z 465.565,A -85,B 0,C 180,E1 -969.225,E2 -969.225} C_VEL
LIN {X 0,Y 594.376,Z 465.573,A -85,B 0,C 180,E1 -972.096,E2 -972.096} C_VEL
LIN {X 0,Y 594.367,Z 465.573,A -85,B 0,C 180,E1 -974.219,E2 -974.219} C_VEL
LIN {X 0,Y 594.364,Z 465.568,A -85,B 0,C 180,E1 -977.017,E2 -977.017} C_VEL
LIN {X 0,Y 594.389,Z 465.572,A -85,B 0,C 180,E1 -979.784,E2 -979.784} C_VEL
LIN {X 0,Y 594.4,Z 465.565,A -85,B 0,C 180,E1 -982.527,E2 -982.527} C_VEL
LIN {X 0,Y 594.385,Z 465.566,A -85,B 0,C 180,E1 -985.252,E2 -985.252} C_VEL
LIN {X 0,Y 594.402,Z 465.573,A -85,B 0,C 180,E1 -987.967,E2 -987.967} C_VEL
LIN {X 0,Y 594.414,Z 465.563,A -85,B 0,C 180,E1 -990.677,E2 -990.677} C_VEL
LIN {X 0,Y 594.379,Z 465.567,A -85,B 0,C 180,E1 -993.389,E2 -993.389} C_VEL
LIN {X 0,Y 594.365,Z 465.577,A -85,B 0,C 180,E1 -996.109,E2 -996.109} C_VEL
LIN {X 0,Y 594.376,Z 465.566,A -85,B 0,C 180,E1 -998.842,E2 -998.842} C_VEL
LIN {X 0,Y 594.392,Z 465.567,A -85,B 0,C 180,E1 -1001.595,E2 -1001.595} C_VEL
LIN {X 0,Y 594.385,Z 465.57,A -85,B 0,C 180,E1 -1004.377,E2 -1004.377} C_VEL
LIN {X 0,Y 594.386,Z 465.565,A -85,B 0,C 180,E1 -1007.193,E2 -1007.193} C_VEL
LIN {X 0,Y 594.373,Z 465.576,A -85,B 0,C 180,E1 -1010.053,E2 -1010.053} C_VEL
LIN {X 0,Y 594.359,Z 465.568,A -85,B 0,C 180,E1 -1012.967,E2 -1012.967} C_VEL
LIN {X 0,Y 594.372,Z 465.566,A -85,B 0,C 180,E1 -1015.193,E2 -1015.193} C_VEL
LIN {X 0,Y 594.379,Z 465.567,A -85,B 0,C 180,E1 -1017.526,E2 -1017.526} C_VEL
LIN {X 0,Y 594.39,Z 465.568,A -85,B 0,C 180,E1 -1020.558,E2 -1020.558} C_VEL
LIN {X 0,Y 594.372,Z 465.567,A -85,B 0,C 180,E1 -1022.95,E2 -1022.95} C_VEL
LIN {X 0,Y 594.374,Z 465.566,A -85,B 0,C 180,E1 -1025.406,E2 -1025.406} C_VEL
LIN {X 0,Y 594.384,Z 465.569,A -85,B 0,C 180,E1 -1027.94,E2 -1027.94} C_VEL
LIN {X 0,Y 594.383,Z 465.566,A -85,B 0,C 180,E1 -1030.823,E2 -1030.823} C_VEL
LIN {X 0,Y 594.379,Z 465.562,A -85,B 0,C 180,E1 -1033.297,E2 -1033.297} C_VEL
LIN {X 0,Y 594.373,Z 465.575,A -85,B 0,C 180,E1 -1036.159,E2 -1036.159} C_VEL
LIN {X 0,Y 594.372,Z 465.565,A -85,B 0,C 180,E1 -1039.177,E2 -1039.177} C_VEL
LIN {X 0,Y 594.379,Z 465.572,A -85,B 0,C 180,E1 -1042.059,E2 -1042.059} C_VEL
LIN {X 0,Y 594.38,Z 465.569,A -85,B 0,C 180,E1 -1044.671,E2 -1044.671} C_VEL
LIN {X 0,Y 594.37,Z 465.567,A -85,B 0,C 180,E1 -1047.088,E2 -1047.088} C_VEL
LIN {X 0,Y 594.391,Z 465.564,A -85,B 0,C 180,E1 -1049.669,E2 -1049.669} C_VEL
LIN {X 0,Y 594.363,Z 465.574,A -85,B 0,C 180,E1 -1052.539,E2 -1052.539} C_VEL
LIN {X 0,Y 594.373,Z 465.568,A -85,B 0,C 180,E1 -1054.807,E2 -1054.807} C_VEL
LIN {X 0,Y 594.355,Z 465.568,A -85,B 0,C 180,E1 -1057.264,E2 -1057.264} C_VEL
LIN {X 0,Y 594.37,Z 465.57,A -85,B 0,C 180,E1 -1059.947,E2 -1059.947} C_VEL
LIN {X 0,Y 594.383,Z 465.568,A -85,B 0,C 180,E1 -1062.807,E2 -1062.807} C_VEL
LIN {X 0,Y 594.378,Z 465.567,A -85,B 0,C 180,E1 -1065.826,E2 -1065.826} C_VEL
LIN {X 0,Y 594.385,Z 465.575,A -85,B 0,C 180,E1 -1068.404,E2 -1068.404} C_VEL
LIN {X 0,Y 594.394,Z 465.563,A -85,B 0,C 180,E1 -1071.158,E2 -1071.158} C_VEL
LIN {X 0,Y 594.362,Z 465.569,A -85,B 0,C 180,E1 -1073.891,E2 -1073.891} C_VEL
LIN {X 0,Y 594.377,Z 465.572,A -85,B 0,C 180,E1 -1076.611,E2 -1076.611} C_VEL
LIN {X 0,Y 594.416,Z 465.56,A -85,B 0,C 180,E1 -1079.323,E2 -1079.323} C_VEL
LIN {X 0,Y 594.388,Z 465.567,A -85,B 0,C 180,E1 -1082.033,E2 -1082.033} C_VEL
LIN {X 0,Y 594.395,Z 465.568,A -85,B 0,C 180,E1 -1084.748,E2 -1084.748} C_VEL
LIN {X 0,Y 594.385,Z 465.564,A -85,B 0,C 180,E1 -1087.474,E2 -1087.474} C_VEL
LIN {X 0,Y 594.388,Z 465.569,A -85,B 0,C 180,E1 -1090.216,E2 -1090.216} C_VEL
LIN {X 0,Y 594.364,Z 465.569,A -85,B 0,C 180,E1 -1092.983,E2 -1092.983} C_VEL
LIN {X 0,Y 594.361,Z 465.567,A -85,B 0,C 180,E1 -1095.781,E2 -1095.781} C_VEL
LIN {X 0,Y 594.382,Z 465.575,A -85,B 0,C 180,E1 -1098.618,E2 -1098.618} C_VEL
LIN {X 0,Y 594.362,Z 465.567,A -85,B 0,C 180,E1 -1101.504,E2 -1101.504} C_VEL
LIN {X 0,Y 594.38,Z 465.573,A -85,B 0,C 180,E1 -1104.447,E2 -1104.447} C_VEL
LIN {X 0,Y 594.379,Z 465.574,A -85,B 0,C 180,E1 -1106.7,E2 -1106.7} C_VEL
LIN {X 0,Y 594.378,Z 465.57,A -85,B 0,C 180,E1 -1108.999,E2 -1108.999} C_VEL
LIN {X 0,Y 594.386,Z 465.564,A -85,B 0,C 180,E1 -1111.646,E2 -1111.646} C_VEL
LIN {X 0,Y 594.393,Z 465.572,A -85,B 0,C 180,E1 -1114.579,E2 -1114.579} C_VEL
LIN {X 0,Y 594.379,Z 465.569,A -85,B 0,C 180,E1 -1117.087,E2 -1117.087} C_VEL
LIN {X 0,Y 594.372,Z 465.566,A -85,B 0,C 180,E1 -1119.775,E2 -1119.775} C_VEL
LIN {X 0,Y 594.362,Z 465.572,A -85,B 0,C 180,E1 -1122.376,E2 -1122.376} C_VEL
LIN {X 0,Y 594.359,Z 465.57,A -85,B 0,C 180,E1 -1125.192,E2 -1125.192} C_VEL
LIN {X 0,Y 594.369,Z 465.566,A -85,B 0,C 180,E1 -1127.626,E2 -1127.626} C_VEL
LIN {X 0,Y 594.387,Z 465.568,A -85,B 0,C 180,E1 -1130.322,E2 -1130.322} C_VEL
LIN {X 0,Y 594.381,Z 465.569,A -85,B 0,C 180,E1 -1132.914,E2 -1132.914} C_VEL
LIN {X 0,Y 594.378,Z 465.566,A -85,B 0,C 180,E1 -1135.862,E2 -1135.862} C_VEL
LIN {X 0,Y 594.389,Z 465.572,A -85,B 0,C 180,E1 -1138.652,E2 -1138.652} C_VEL
LIN {X 0,Y 594.381,Z 465.572,A -85,B 0,C 180,E1 -1141.043,E2 -1141.043} C_VEL
LIN {X 0,Y 594.381,Z 465.57,A -85,B 0,C 180,E1 -1143.979,E2 -1143.979} C_VEL
LIN {X 0,Y 594.413,Z 465.79,A -85,B 0,C 180,E1 -1144.458,E2 -1144.458} C_VEL
LIN {X 0,Y 594.803,Z 469.192,A -85,B 0,C 180,E1 -1145.032,E2 -1145.032} C_VEL
LIN {X 0,Y 594.688,Z 486.519,A -85,B 0,C 180,E1 -1147.78,E2 -1147.78} C_VEL
LIN {X 0,Y 594.593,Z 505.125,A -85,B 0,C 180,E1 -1150.674,E2 -1150.674} C_VEL
LIN {X 0,Y 594.505,Z 523.731,A -85,B 0,C 180,E1 -1153.518,E2 -1153.518} C_VEL
LIN {X 0,Y 594.523,Z 526.256,A -85,B 0,C 180,E1 -1153.849,E2 -1153.849} C_VEL
LIN {X 0,Y 595.014,Z 530.435,A -85,B 0,C 180,E1 -1153.929,E2 -1153.929} C_VEL
LIN {X 0,Y 594.858,Z 662.881,A -85,B 0,C 180,E1 -1155.569,E2 -1155.569} C_VEL
LIN {X 0,Y 594.801,Z 677.757,A -85,B 0,C 180,E1 -1155.905,E2 -1155.905} C_VEL
LIN {X 0,Y 594.755,Z 691.84,A -85,B 0,C 180,E1 -1156.374,E2 -1156.374} C_VEL
LIN {X 0,Y 594.653,Z 704.605,A -85,B 0,C 180,E1 -1156.937,E2 -1156.937} C_VEL
LIN {X 0,Y 594.572,Z 717.095,A -85,B 0,C 180,E1 -1157.629,E2 -1157.629} C_VEL
LIN {X 0,Y 594.524,Z 729.563,A -85,B 0,C 180,E1 -1158.487,E2 -1158.487} C_VEL
LIN {X 0,Y 594.449,Z 740.817,A -85,B 0,C 180,E1 -1159.441,E2 -1159.441} C_VEL
LIN {X 0,Y 594.368,Z 750.855,A -85,B 0,C 180,E1 -1160.472,E2 -1160.472} C_VEL
LIN {X 0,Y 594.346,Z 760.414,A -85,B 0,C 180,E1 -1161.671,E2 -1161.671} C_VEL
LIN {X 0,Y 594.303,Z 768.142,A -85,B 0,C 180,E1 -1162.867,E2 -1162.867} C_VEL
LIN {X 0,Y 594.279,Z 773.525,A -85,B 0,C 180,E1 -1163.89,E2 -1163.89} C_VEL
LIN {X 0,Y 594.247,Z 777.949,A -85,B 0,C 180,E1 -1164.911,E2 -1164.911} C_VEL
LIN {X 0,Y 594.259,Z 781.446,A -85,B 0,C 180,E1 -1165.931,E2 -1165.931} C_VEL
LIN {X 0,Y 594.224,Z 784.828,A -85,B 0,C 180,E1 -1167.288,E2 -1167.288} C_VEL
LIN {X 0,Y 594.241,Z 786.823,A -85,B 0,C 180,E1 -1168.645,E2 -1168.645} C_VEL
LIN {X 0,Y 594.234,Z 787.5,A -85,B 0,C 180,E1 -1170,E2 -1170} C_VEL
LIN {X 0,Y 594.241,Z 786.823,A -85,B 0,C 180,E1 -1171.355,E2 -1171.355} C_VEL
LIN {X 0,Y 594.224,Z 784.828,A -85,B 0,C 180,E1 -1172.712,E2 -1172.712} C_VEL
LIN {X 0,Y 594.259,Z 781.446,A -85,B 0,C 180,E1 -1174.069,E2 -1174.069} C_VEL
LIN {X 0,Y 594.275,Z 776.574,A -85,B 0,C 180,E1 -1175.429,E2 -1175.429} C_VEL
LIN {X 0,Y 594.277,Z 770.054,A -85,B 0,C 180,E1 -1176.792,E2 -1176.792} C_VEL
LIN {X 0,Y 594.329,Z 762.787,A -85,B 0,C 180,E1 -1177.987,E2 -1177.987} C_VEL
LIN {X 0,Y 594.367,Z 753.826,A -85,B 0,C 180,E1 -1179.185,E2 -1179.185} C_VEL
LIN {X 0,Y 594.411,Z 744.387,A -85,B 0,C 180,E1 -1180.215,E2 -1180.215} C_VEL
LIN {X 0,Y 594.509,Z 734.295,A -85,B 0,C 180,E1 -1181.131,E2 -1181.131} C_VEL
LIN {X 0,Y 594.569,Z 723.702,A -85,B 0,C 180,E1 -1181.938,E2 -1181.938} C_VEL
LIN {X 0,Y 594.616,Z 711.226,A -85,B 0,C 180,E1 -1182.717,E2 -1182.717} C_VEL
LIN {X 0,Y 594.706,Z 697.18,A -85,B 0,C 180,E1 -1183.41,E2 -1183.41} C_VEL
LIN {X 0,Y 594.787,Z 685.185,A -85,B 0,C 180,E1 -1183.866,E2 -1183.866} C_VEL
LIN {X 0,Y 594.816,Z 671.637,A -85,B 0,C 180,E1 -1184.25,E2 -1184.25} C_VEL
LIN {X 0,Y 594.897,Z 658.651,A -85,B 0,C 180,E1 -1184.495,E2 -1184.495} C_VEL
LIN {X 0,Y 594.879,Z 528.198,A -85,B 0,C 180,E1 -1186.102,E2 -1186.102} C_VEL
LIN {X 0,Y 594.501,Z 525.915,A -85,B 0,C 180,E1 -1186.173,E2 -1186.173} C_VEL
LIN {X 0,Y 594.561,Z 510.939,A -85,B 0,C 180,E1 -1188.433,E2 -1188.433} C_VEL
LIN {X 0,Y 594.646,Z 493.164,A -85,B 0,C 180,E1 -1191.181,E2 -1191.181} C_VEL
LIN {X 0,Y 594.745,Z 476.053,A -85,B 0,C 180,E1 -1193.873,E2 -1193.873} C_VEL
LIN {X 0,Y 594.771,Z 467.913,A -85,B 0,C 180,E1 -1195.175,E2 -1195.175} C_VEL
LIN {X 0,Y 594.412,Z 465.631,A -85,B 0,C 180,E1 -1195.613,E2 -1195.613} C_VEL
LIN {X 0,Y 594.374,Z 465.566,A -85,B 0,C 180,E1 -1198.226,E2 -1198.226} C_VEL
LIN {X 0,Y 594.387,Z 465.566,A -85,B 0,C 180,E1 -1200.558,E2 -1200.558} C_VEL
LIN {X 0,Y 594.377,Z 465.572,A -85,B 0,C 180,E1 -1202.949,E2 -1202.949} C_VEL
LIN {X 0,Y 594.346,Z 465.573,A -85,B 0,C 180,E1 -1205.408,E2 -1205.408} C_VEL
LIN {X 0,Y 594.386,Z 465.564,A -85,B 0,C 180,E1 -1207.94,E2 -1207.94} C_VEL
LIN {X 0,Y 594.376,Z 465.57,A -85,B 0,C 180,E1 -1210.822,E2 -1210.822} C_VEL
LIN {X 0,Y 594.378,Z 465.566,A -85,B 0,C 180,E1 -1213.84,E2 -1213.84} C_VEL
LIN {X 0,Y 594.361,Z 465.57,A -85,B 0,C 180,E1 -1216.7,E2 -1216.7} C_VEL
LIN {X 0,Y 594.365,Z 465.575,A -85,B 0,C 180,E1 -1219.432,E2 -1219.432} C_VEL
LIN {X 0,Y 594.383,Z 465.564,A -85,B 0,C 180,E1 -1222.391,E2 -1222.391} C_VEL
LIN {X 0,Y 594.382,Z 465.566,A -85,B 0,C 180,E1 -1224.671,E2 -1224.671} C_VEL
LIN {X 0,Y 594.373,Z 465.572,A -85,B 0,C 180,E1 -1227.087,E2 -1227.087} C_VEL
LIN {X 0,Y 594.38,Z 465.57,A -85,B 0,C 180,E1 -1229.671,E2 -1229.671} C_VEL
LIN {X 0,Y 594.366,Z 465.566,A -85,B 0,C 180,E1 -1232.538,E2 -1232.538} C_VEL
LIN {X 0,Y 594.374,Z 465.568,A -85,B 0,C 180,E1 -1234.807,E2 -1234.807} C_VEL
LIN {X 0,Y 594.357,Z 465.577,A -85,B 0,C 180,E1 -1237.264,E2 -1237.264} C_VEL
LIN {X 0,Y 594.37,Z 465.568,A -85,B 0,C 180,E1 -1239.946,E2 -1239.946} C_VEL
LIN {X 0,Y 594.383,Z 465.566,A -85,B 0,C 180,E1 -1242.806,E2 -1242.806} C_VEL
LIN {X 0,Y 594.379,Z 465.568,A -85,B 0,C 180,E1 -1245.825,E2 -1245.825} C_VEL
LIN {X 0,Y 594.386,Z 465.564,A -85,B 0,C 180,E1 -1248.404,E2 -1248.404} C_VEL
LIN {X 0,Y 594.394,Z 465.569,A -85,B 0,C 180,E1 -1251.158,E2 -1251.158} C_VEL
LIN {X 0,Y 594.362,Z 465.569,A -85,B 0,C 180,E1 -1253.891,E2 -1253.891} C_VEL
LIN {X 0,Y 594.377,Z 465.565,A -85,B 0,C 180,E1 -1256.61,E2 -1256.61} C_VEL
LIN {X 0,Y 594.417,Z 465.568,A -85,B 0,C 180,E1 -1259.322,E2 -1259.322} C_VEL
LIN {X 0,Y 594.388,Z 465.565,A -85,B 0,C 180,E1 -1262.032,E2 -1262.032} C_VEL
LIN {X 0,Y 594.396,Z 465.563,A -85,B 0,C 180,E1 -1264.747,E2 -1264.747} C_VEL
LIN {X 0,Y 594.393,Z 465.573,A -85,B 0,C 180,E1 -1267.473,E2 -1267.473} C_VEL
LIN {X 0,Y 594.388,Z 465.564,A -85,B 0,C 180,E1 -1270.216,E2 -1270.216} C_VEL
LIN {X 0,Y 594.364,Z 465.569,A -85,B 0,C 180,E1 -1272.983,E2 -1272.983} C_VEL
LIN {X 0,Y 594.355,Z 465.571,A -85,B 0,C 180,E1 -1275.34,E2 -1275.34} C_VEL
LIN {X 0,Y 593.685,Z 465.658,A -85,B 0,C 180,E1 -1275.905,E2 -1275.905} C_VEL
LIN {X 0,Y 590.831,Z 466.013,A -85,B 0,C 180,E1 -1276.824,E2 -1276.824} C_VEL
LIN {X 0,Y 588.426,Z 466.315,A -85,B 0,C 180,E1 -1277.562,E2 -1277.562} C_VEL
LIN {X 0,Y 587.399,Z 466.436,A -85,B 0,C 180,E1 -1278.132,E2 -1278.132} C_VEL
LIN {X 0,Y 587.318,Z 466.445,A -85,B 0,C 180,E1 -1278.325,E2 -1278.325} C_VEL
LIN {X 0,Y 587.347,Z 466.443,A -85,B 0,C 180,E1 -1281.045,E2 -1281.045} C_VEL
LIN {X 0,Y 587.328,Z 466.446,A -85,B 0,C 180,E1 -1284.006,E2 -1284.006} C_VEL
LIN {X 0,Y 587.355,Z 466.442,A -85,B 0,C 180,E1 -1286.277,E2 -1286.277} C_VEL
LIN {X 0,Y 587.345,Z 466.444,A -85,B 0,C 180,E1 -1289.135,E2 -1289.135} C_VEL
LIN {X 0,Y 587.348,Z 466.449,A -85,B 0,C 180,E1 -1291.838,E2 -1291.838} C_VEL
LIN {X 0,Y 587.35,Z 466.442,A -85,B 0,C 180,E1 -1294.35,E2 -1294.35} C_VEL
LIN {X 0,Y 587.344,Z 466.441,A -85,B 0,C 180,E1 -1296.747,E2 -1296.747} C_VEL
LIN {X 0,Y 587.34,Z 466.447,A -85,B 0,C 180,E1 -1299.359,E2 -1299.359} C_VEL
LIN {X 0,Y 587.325,Z 466.449,A -85,B 0,C 180,E1 -1302.108,E2 -1302.108} C_VEL
LIN {X 0,Y 587.307,Z 466.447,A -85,B 0,C 180,E1 -1305.089,E2 -1305.089} C_VEL
LIN {X 0,Y 587.344,Z 466.449,A -85,B 0,C 180,E1 -1307.928,E2 -1307.928} C_VEL
LIN {X 0,Y 587.34,Z 466.443,A -85,B 0,C 180,E1 -1310.641,E2 -1310.641} C_VEL
LIN {X 0,Y 587.347,Z 466.442,A -85,B 0,C 180,E1 -1313.292,E2 -1313.292} C_VEL
LIN {X 0,Y 587.359,Z 466.45,A -85,B 0,C 180,E1 -1315.781,E2 -1315.781} C_VEL
LIN {X 0,Y 587.348,Z 466.445,A -85,B 0,C 180,E1 -1318.232,E2 -1318.232} C_VEL
LIN {X 0,Y 587.344,Z 466.442,A -85,B 0,C 180,E1 -1320.867,E2 -1320.867} C_VEL
LIN {X 0,Y 587.354,Z 466.451,A -85,B 0,C 180,E1 -1323.819,E2 -1323.819} C_VEL
LIN {X 0,Y 587.335,Z 466.452,A -85,B 0,C 180,E1 -1325.994,E2 -1325.994} C_VEL
LIN {X 0,Y 587.319,Z 466.45,A -85,B 0,C 180,E1 -1328.226,E2 -1328.226} C_VEL
LIN {X 0,Y 587.344,Z 466.443,A -85,B 0,C 180,E1 -1331.151,E2 -1331.151} C_VEL
LIN {X 0,Y 587.346,Z 466.444,A -85,B 0,C 180,E1 -1333.311,E2 -1333.311} C_VEL
LIN {X 0,Y 587.357,Z 466.447,A -85,B 0,C 180,E1 -1336.155,E2 -1336.155} C_VEL
LIN {X 0,Y 587.338,Z 466.443,A -85,B 0,C 180,E1 -1338.963,E2 -1338.963} C_VEL
LIN {X 0,Y 587.362,Z 466.447,A -85,B 0,C 180,E1 -1341.745,E2 -1341.745} C_VEL
LIN {X 0,Y 587.353,Z 466.443,A -85,B 0,C 180,E1 -1344.507,E2 -1344.507} C_VEL
LIN {X 0,Y 587.368,Z 466.44,A -85,B 0,C 180,E1 -1347.257,E2 -1347.257} C_VEL
LIN {X 0,Y 587.382,Z 466.448,A -85,B 0,C 180,E1 -1350,E2 -1350} C_VEL
LIN {X 0,Y 587.368,Z 466.44,A -85,B 0,C 180,E1 -1352.743,E2 -1352.743} C_VEL
LIN {X 0,Y 587.355,Z 466.443,A -85,B 0,C 180,E1 -1355.493,E2 -1355.493} C_VEL
LIN {X 0,Y 587.362,Z 466.447,A -85,B 0,C 180,E1 -1358.255,E2 -1358.255} C_VEL
LIN {X 0,Y 587.344,Z 466.442,A -85,B 0,C 180,E1 -1361.133,E2 -1361.133} C_VEL
LIN {X 0,Y 587.361,Z 466.448,A -85,B 0,C 180,E1 -1364.26,E2 -1364.26} C_VEL
LIN {X 0,Y 587.354,Z 466.442,A -85,B 0,C 180,E1 -1367.405,E2 -1367.405} C_VEL
LIN {X 0,Y 587.326,Z 466.452,A -85,B 0,C 180,E1 -1370.304,E2 -1370.304} C_VEL
LIN {X 0,Y 587.319,Z 466.445,A -85,B 0,C 180,E1 -1373.258,E2 -1373.258} C_VEL
LIN {X 0,Y 587.33,Z 466.445,A -85,B 0,C 180,E1 -1375.516,E2 -1375.516} C_VEL
LIN {X 0,Y 587.343,Z 466.447,A -85,B 0,C 180,E1 -1377.817,E2 -1377.817} C_VEL
LIN {X 0,Y 587.346,Z 466.447,A -85,B 0,C 180,E1 -1380.512,E2 -1380.512} C_VEL
LIN {X 0,Y 587.329,Z 466.444,A -85,B 0,C 180,E1 -1383.396,E2 -1383.396} C_VEL
LIN {X 0,Y 587.348,Z 466.446,A -85,B 0,C 180,E1 -1385.895,E2 -1385.895} C_VEL
LIN {X 0,Y 587.328,Z 466.45,A -85,B 0,C 180,E1 -1388.478,E2 -1388.478} C_VEL
LIN {X 0,Y 587.334,Z 466.442,A -85,B 0,C 180,E1 -1391.156,E2 -1391.156} C_VEL
LIN {X 0,Y 587.326,Z 466.448,A -85,B 0,C 180,E1 -1394.114,E2 -1394.114} C_VEL
LIN {X 0,Y 587.312,Z 466.447,A -85,B 0,C 180,E1 -1396.994,E2 -1396.994} C_VEL
LIN {X 0,Y 587.313,Z 466.447,A -85,B 0,C 180,E1 -1399.746,E2 -1399.746} C_VEL
LIN {X 0,Y 587.336,Z 466.451,A -85,B 0,C 180,E1 -1402.392,E2 -1402.392} C_VEL
LIN {X 0,Y 587.345,Z 466.443,A -85,B 0,C 180,E1 -1404.946,E2 -1404.946} C_VEL
LIN {X 0,Y 587.332,Z 466.443,A -85,B 0,C 180,E1 -1407.421,E2 -1407.421} C_VEL
LIN {X 0,Y 587.337,Z 466.444,A -85,B 0,C 180,E1 -1409.831,E2 -1409.831} C_VEL
LIN {X 0,Y 587.341,Z 466.452,A -85,B 0,C 180,E1 -1412.307,E2 -1412.307} C_VEL
LIN {X 0,Y 587.333,Z 466.45,A -85,B 0,C 180,E1 -1414.484,E2 -1414.484} C_VEL
LIN {X 0,Y 587.331,Z 466.443,A -85,B 0,C 180,E1 -1417.486,E2 -1417.486} C_VEL
LIN {X 0,Y 587.325,Z 466.445,A -85,B 0,C 180,E1 -1419.695,E2 -1419.695} C_VEL
LIN {X 0,Y 587.35,Z 466.447,A -85,B 0,C 180,E1 -1422.594,E2 -1422.594} C_VEL
LIN {X 0,Y 587.354,Z 466.441,A -85,B 0,C 180,E1 -1425.739,E2 -1425.739} C_VEL
LIN {X 0,Y 587.351,Z 466.443,A -85,B 0,C 180,E1 -1428.859,E2 -1428.859} C_VEL
LIN {X 0,Y 587.363,Z 466.439,A -85,B 0,C 180,E1 -1431.745,E2 -1431.745} C_VEL
LIN {X 0,Y 587.351,Z 466.45,A -85,B 0,C 180,E1 -1434.507,E2 -1434.507} C_VEL
LIN {X 0,Y 587.374,Z 466.436,A -85,B 0,C 180,E1 -1437.257,E2 -1437.257} C_VEL
LIN {X 0,Y 587.373,Z 466.44,A -85,B 0,C 180,E1 -1440,E2 -1440} C_VEL
LIN {X 0,Y 587.374,Z 466.444,A -85,B 0,C 180,E1 -1442.744,E2 -1442.744} C_VEL
LIN {X 0,Y 587.351,Z 466.438,A -85,B 0,C 180,E1 -1445.493,E2 -1445.493} C_VEL
LIN {X 0,Y 587.364,Z 466.444,A -85,B 0,C 180,E1 -1448.256,E2 -1448.256} C_VEL
LIN {X 0,Y 587.337,Z 466.444,A -85,B 0,C 180,E1 -1451.134,E2 -1451.134} C_VEL
LIN {X 0,Y 587.35,Z 466.439,A -85,B 0,C 180,E1 -1453.846,E2 -1453.846} C_VEL
LIN {X 0,Y 587.353,Z 466.447,A -85,B 0,C 180,E1 -1456.82,E2 -1456.82} C_VEL
LIN {X 0,Y 587.336,Z 466.441,A -85,B 0,C 180,E1 -1459.576,E2 -1459.576} C_VEL
LIN {X 0,Y 587.316,Z 466.444,A -85,B 0,C 180,E1 -1461.775,E2 -1461.775} C_VEL
LIN {X 0,Y 587.345,Z 466.449,A -85,B 0,C 180,E1 -1464.759,E2 -1464.759} C_VEL
LIN {X 0,Y 587.322,Z 466.447,A -85,B 0,C 180,E1 -1467.047,E2 -1467.047} C_VEL
LIN {X 0,Y 587.342,Z 466.443,A -85,B 0,C 180,E1 -1469.38,E2 -1469.38} C_VEL
LIN {X 0,Y 587.349,Z 466.441,A -85,B 0,C 180,E1 -1471.838,E2 -1471.838} C_VEL
LIN {X 0,Y 587.351,Z 466.445,A -85,B 0,C 180,E1 -1474.35,E2 -1474.35} C_VEL
LIN {X 0,Y 587.347,Z 466.451,A -85,B 0,C 180,E1 -1476.747,E2 -1476.747} C_VEL
LIN {X 0,Y 587.342,Z 466.443,A -85,B 0,C 180,E1 -1479.36,E2 -1479.36} C_VEL
LIN {X 0,Y 587.329,Z 466.445,A -85,B 0,C 180,E1 -1482.109,E2 -1482.109} C_VEL
LIN {X 0,Y 587.312,Z 466.449,A -85,B 0,C 180,E1 -1485.09,E2 -1485.09} C_VEL
LIN {X 0,Y 587.349,Z 466.44,A -85,B 0,C 180,E1 -1487.928,E2 -1487.928} C_VEL
LIN {X 0,Y 587.331,Z 466.447,A -85,B 0,C 180,E1 -1491.059,E2 -1491.059} C_VEL
LIN {X 0,Y 587.345,Z 466.439,A -85,B 0,C 180,E1 -1493.293,E2 -1493.293} C_VEL
LIN {X 0,Y 587.358,Z 466.44,A -85,B 0,C 180,E1 -1495.781,E2 -1495.781} C_VEL
LIN {X 0,Y 587.351,Z 466.442,A -85,B 0,C 180,E1 -1498.233,E2 -1498.233} C_VEL
LIN {X 0,Y 587.348,Z 466.452,A -85,B 0,C 180,E1 -1500.867,E2 -1500.867} C_VEL
LIN {X 0,Y 587.357,Z 466.447,A -85,B 0,C 180,E1 -1503.82,E2 -1503.82} C_VEL
LIN {X 0,Y 587.367,Z 466.575,A -85,B 0,C 180,E1 -1504.248,E2 -1504.248} C_VEL
LIN {X 0,Y 587.904,Z 470.238,A -85,B 0,C 180,E1 -1504.889,E2 -1504.889} C_VEL
LIN {X 0,Y 587.746,Z 487.682,A -85,B 0,C 180,E1 -1507.688,E2 -1507.688} C_VEL
LIN {X 0,Y 587.596,Z 505.125,A -85,B 0,C 180,E1 -1510.434,E2 -1510.434} C_VEL
LIN {X 0,Y 587.537,Z 521.207,A -85,B 0,C 180,E1 -1512.928,E2 -1512.928} C_VEL
LIN {X 0,Y 587.529,Z 525.911,A -85,B 0,C 180,E1 -1513.63,E2 -1513.63} C_VEL
LIN {X 0,Y 588.076,Z 529.217,A -85,B 0,C 180,E1 -1513.719,E2 -1513.719} C_VEL
LIN {X 0,Y 588.029,Z 661.475,A -85,B 0,C 180,E1 -1515.376,E2 -1515.376} C_VEL
LIN {X 0,Y 587.916,Z 675.855,A -85,B 0,C 180,E1 -1515.682,E2 -1515.682} C_VEL
LIN {X 0,Y 587.843,Z 690.719,A -85,B 0,C 180,E1 -1516.166,E2 -1516.166} C_VEL
LIN {X 0,Y 587.758,Z 702.845,A -85,B 0,C 180,E1 -1516.693,E2 -1516.693} C_VEL
LIN {X 0,Y 587.654,Z 714.229,A -85,B 0,C 180,E1 -1517.306,E2 -1517.306} C_VEL
LIN {X 0,Y 587.55,Z 726.16,A -85,B 0,C 180,E1 -1518.093,E2 -1518.093} C_VEL
LIN {X 0,Y 587.464,Z 737.008,A -85,B 0,C 180,E1 -1518.965,E2 -1518.965} C_VEL
LIN {X 0,Y 587.344,Z 747.716,A -85,B 0,C 180,E1 -1520.009,E2 -1520.009} C_VEL
LIN {X 0,Y 587.312,Z 756.553,A -85,B 0,C 180,E1 -1521.051,E2 -1521.051} C_VEL
LIN {X 0,Y 587.261,Z 763.906,A -85,B 0,C 180,E1 -1522.09,E2 -1522.09} C_VEL
LIN {X 0,Y 587.209,Z 770.055,A -85,B 0,C 180,E1 -1523.126,E2 -1523.126} C_VEL
LIN {X 0,Y 587.199,Z 776.577,A -85,B 0,C 180,E1 -1524.506,E2 -1524.506} C_VEL
LIN {X 0,Y 587.179,Z 781.448,A -85,B 0,C 180,E1 -1525.882,E2 -1525.882} C_VEL
LIN {X 0,Y 587.13,Z 784.821,A -85,B 0,C 180,E1 -1527.256,E2 -1527.256} C_VEL
LIN {X 0,Y 587.141,Z 786.82,A -85,B 0,C 180,E1 -1528.628,E2 -1528.628} C_VEL
LIN {X 0,Y 587.135,Z 787.5,A -85,B 0,C 180,E1 -1530,E2 -1530} C_VEL
LIN {X 0,Y 587.141,Z 786.82,A -85,B 0,C 180,E1 -1531.372,E2 -1531.372} C_VEL
LIN {X 0,Y 587.13,Z 784.821,A -85,B 0,C 180,E1 -1532.744,E2 -1532.744} C_VEL
LIN {X 0,Y 587.179,Z 781.448,A -85,B 0,C 180,E1 -1534.118,E2 -1534.118} C_VEL
LIN {X 0,Y 587.199,Z 776.577,A -85,B 0,C 180,E1 -1535.494,E2 -1535.494} C_VEL
LIN {X 0,Y 587.209,Z 770.055,A -85,B 0,C 180,E1 -1536.874,E2 -1536.874} C_VEL
LIN {X 0,Y 587.268,Z 762.781,A -85,B 0,C 180,E1 -1538.083,E2 -1538.083} C_VEL
LIN {X 0,Y 587.322,Z 753.826,A -85,B 0,C 180,E1 -1539.296,E2 -1539.296} C_VEL
LIN {X 0,Y 587.372,Z 744.384,A -85,B 0,C 180,E1 -1540.339,E2 -1540.339} C_VEL
LIN {X 0,Y 587.471,Z 733.992,A -85,B 0,C 180,E1 -1541.291,E2 -1541.291} C_VEL
LIN {X 0,Y 587.576,Z 723.691,A -85,B 0,C 180,E1 -1542.082,E2 -1542.082} C_VEL
LIN {X 0,Y 587.646,Z 711.231,A -85,B 0,C 180,E1 -1542.87,E2 -1542.87} C_VEL
LIN {X 0,Y 587.787,Z 697.186,A -85,B 0,C 180,E1 -1543.571,E2 -1543.571} C_VEL
LIN {X 0,Y 587.911,Z 683.583,A -85,B 0,C 180,E1 -1544.085,E2 -1544.085} C_VEL
LIN {X 0,Y 587.953,Z 670.358,A -85,B 0,C 180,E1 -1544.45,E2 -1544.45} C_VEL
LIN {X 0,Y 588.014,Z 655.627,A -85,B 0,C 180,E1 -1544.713,E2 -1544.713} C_VEL
LIN {X 0,Y 588.063,Z 529.095,A -85,B 0,C 180,E1 -1546.283,E2 -1546.283} C_VEL
LIN {X 0,Y 587.529,Z 525.912,A -85,B 0,C 180,E1 -1546.37,E2 -1546.37} C_VEL
LIN {X 0,Y 587.582,Z 508.07,A -85,B 0,C 180,E1 -1549.106,E2 -1549.106} C_VEL
LIN {X 0,Y 587.751,Z 490.007,A -85,B 0,C 180,E1 -1551.942,E2 -1551.942} C_VEL
LIN {X 0,Y 587.899,Z 472.564,A -85,B 0,C 180,E1 -1554.733,E2 -1554.733} C_VEL
LIN {X 0,Y 587.641,Z 467.913,A -85,B 0,C 180,E1 -1555.502,E2 -1555.502} C_VEL
LIN {X 0,Y 587.374,Z 466.509,A -85,B 0,C 180,E1 -1555.799,E2 -1555.799} C_VEL
LIN {X 0,Y 587.321,Z 466.447,A -85,B 0,C 180,E1 -1558.596,E2 -1558.596} C_VEL
LIN {X 0,Y 587.34,Z 466.447,A -85,B 0,C 180,E1 -1560.965,E2 -1560.965} C_VEL
LIN {X 0,Y 587.333,Z 466.451,A -85,B 0,C 180,E1 -1563.396,E2 -1563.396} C_VEL
LIN {X 0,Y 587.288,Z 466.445,A -85,B 0,C 180,E1 -1565.899,E2 -1565.899} C_VEL
LIN {X 0,Y 587.331,Z 466.442,A -85,B 0,C 180,E1 -1568.478,E2 -1568.478} C_VEL
LIN {X 0,Y 587.334,Z 466.453,A -85,B 0,C 180,E1 -1571.156,E2 -1571.156} C_VEL
LIN {X 0,Y 587.33,Z 466.442,A -85,B 0,C 180,E1 -1574.113,E2 -1574.113} C_VEL
LIN {X 0,Y 587.309,Z 466.452,A -85,B 0,C 180,E1 -1576.993,E2 -1576.993} C_VEL
LIN {X 0,Y 587.314,Z 466.449,A -85,B 0,C 180,E1 -1579.745,E2 -1579.745} C_VEL
LIN {X 0,Y 587.338,Z 466.442,A -85,B 0,C 180,E1 -1582.392,E2 -1582.392} C_VEL
LIN {X 0,Y 587.346,Z 466.446,A -85,B 0,C 180,E1 -1584.945,E2 -1584.945} C_VEL
LIN {X 0,Y 587.334,Z 466.452,A -85,B 0,C 180,E1 -1587.42,E2 -1587.42} C_VEL
LIN {X 0,Y 587.328,Z 466.447,A -85,B 0,C 180,E1 -1589.829,E2 -1589.829} C_VEL
LIN {X 0,Y 587.344,Z 466.44,A -85,B 0,C 180,E1 -1592.306,E2 -1592.306} C_VEL
LIN {X 0,Y 587.334,Z 466.442,A -85,B 0,C 180,E1 -1594.483,E2 -1594.483} C_VEL
LIN {X 0,Y 587.333,Z 466.451,A -85,B 0,C 180,E1 -1597.486,E2 -1597.486} C_VEL
LIN {X 0,Y 587.325,Z 466.448,A -85,B 0,C 180,E1 -1599.695,E2 -1599.695} C_VEL
LIN {X 0,Y 587.35,Z 466.441,A -85,B 0,C 180,E1 -1602.594,E2 -1602.594} C_VEL
LIN {X 0,Y 587.355,Z 466.443,A -85,B 0,C 180,E1 -1605.739,E2 -1605.739} C_VEL
LIN {X 0,Y 587.334,Z 466.443,A -85,B 0,C 180,E1 -1608.263,E2 -1608.263} C_VEL
LIN {X 0,Y 587.338,Z 466.446,A -85,B 0,C 180,E1 -1611.051,E2 -1611.051} C_VEL
LIN {X 0,Y 587.365,Z 466.445,A -85,B 0,C 180,E1 -1613.264,E2 -1613.264} C_VEL
LIN {X 0,Y 587.31,Z 466.449,A -85,B 0,C 180,E1 -1615.882,E2 -1615.882} C_VEL
LIN {X 0,Y 587.359,Z 466.443,A -85,B 0,C 180,E1 -1617.943,E2 -1617.943} C_VEL
LIN {X 0,Y 587.389,Z 466.435,A -85,B 0,C 180,E1 -1620.685,E2 -1620.685} C_VEL
LIN {X 0,Y 587.329,Z 466.45,A -85,B 0,C 180,E1 -1623.43,E2 -1623.43} C_VEL
LIN {X 0,Y 587.349,Z 466.451,A -85,B 0,C 180,E1 -1625.493,E2 -1625.493} C_VEL
LIN {X 0,Y 587.363,Z 466.439,A -85,B 0,C 180,E1 -1628.255,E2 -1628.255} C_VEL
LIN {X 0,Y 587.351,Z 466.443,A -85,B 0,C 180,E1 -1631.141,E2 -1631.141} C_VEL
LIN {X 0,Y 587.354,Z 466.441,A -85,B 0,C 180,E1 -1634.261,E2 -1634.261} C_VEL
LIN {X 0,Y 587.35,Z 466.447,A -85,B 0,C 180,E1 -1637.406,E2 -1637.406} C_VEL
LIN {X 0,Y 587.318,Z 466.445,A -85,B 0,C 180,E1 -1638.325,E2 -1638.325} C_VEL
LIN {X 0,Y 586.666,Z 466.526,A -85,B 0,C 180,E1 -1638.897,E2 -1638.897} C_VEL
LIN {X 0,Y 583.835,Z 466.886,A -85,B 0,C 180,E1 -1639.826,E2 -1639.826} C_VEL
LIN {X 0,Y 581.425,Z 467.188,A -85,B 0,C 180,E1 -1640.573,E2 -1640.573} C_VEL
LIN {X 0,Y 580.372,Z 467.317,A -85,B 0,C 180,E1 -1641.149,E2 -1641.149} C_VEL
LIN {X 0,Y 580.277,Z 467.327,A -85,B 0,C 180,E1 -1641.344,E2 -1641.344} C_VEL
LIN {X 0,Y 580.291,Z 467.319,A -85,B 0,C 180,E1 -1644.316,E2 -1644.316} C_VEL
LIN {X 0,Y 580.298,Z 467.319,A -85,B 0,C 180,E1 -1646.622,E2 -1646.622} C_VEL
LIN {X 0,Y 580.299,Z 467.324,A -85,B 0,C 180,E1 -1649.311,E2 -1649.311} C_VEL
LIN {X 0,Y 580.294,Z 467.322,A -85,B 0,C 180,E1 -1652.2,E2 -1652.2} C_VEL
LIN {X 0,Y 580.294,Z 467.319,A -85,B 0,C 180,E1 -1654.695,E2 -1654.695} C_VEL
LIN {X 0,Y 580.291,Z 467.323,A -85,B 0,C 180,E1 -1657.268,E2 -1657.268} C_VEL
LIN {X 0,Y 580.291,Z 467.321,A -85,B 0,C 180,E1 -1660.272,E2 -1660.272} C_VEL
LIN {X 0,Y 580.272,Z 467.323,A -85,B 0,C 180,E1 -1662.706,E2 -1662.706} C_VEL
LIN {X 0,Y 580.265,Z 467.331,A -85,B 0,C 180,E1 -1665.609,E2 -1665.609} C_VEL
LIN {X 0,Y 580.313,Z 467.32,A -85,B 0,C 180,E1 -1668.235,E2 -1668.235} C_VEL
LIN {X 0,Y 580.284,Z 467.322,A -85,B 0,C 180,E1 -1670.967,E2 -1670.967} C_VEL
LIN {X 0,Y 580.29,Z 467.325,A -85,B 0,C 180,E1 -1673.599,E2 -1673.599} C_VEL
LIN {X 0,Y 580.312,Z 467.323,A -85,B 0,C 180,E1 -1676.146,E2 -1676.146} C_VEL
LIN {X 0,Y 580.284,Z 467.322,A -85,B 0,C 180,E1 -1678.616,E2 -1678.616} C_VEL
LIN {X 0,Y 580.288,Z 467.321,A -85,B 0,C 180,E1 -1681.024,E2 -1681.024} C_VEL
LIN {X 0,Y 580.286,Z 467.329,A -85,B 0,C 180,E1 -1683.666,E2 -1683.666} C_VEL
LIN {X 0,Y 580.297,Z 467.328,A -85,B 0,C 180,E1 -1685.684,E2 -1685.684} C_VEL
LIN {X 0,Y 580.27,Z 467.333,A -85,B 0,C 180,E1 -1687.948,E2 -1687.948} C_VEL
LIN {X 0,Y 580.314,Z 467.318,A -85,B 0,C 180,E1 -1690.914,E2 -1690.914} C_VEL
LIN {X 0,Y 580.277,Z 467.332,A -85,B 0,C 180,E1 -1693.826,E2 -1693.826} C_VEL
LIN {X 0,Y 580.323,Z 467.327,A -85,B 0,C 180,E1 -1695.983,E2 -1695.983} C_VEL
LIN {X 0,Y 580.301,Z 467.32,A -85,B 0,C 180,E1 -1698.827,E2 -1698.827} C_VEL
LIN {X 0,Y 580.325,Z 467.322,A -85,B 0,C 180,E1 -1701.644,E2 -1701.644} C_VEL
LIN {X 0,Y 580.319,Z 467.321,A -85,B 0,C 180,E1 -1704.44,E2 -1704.44} C_VEL
LIN {X 0,Y 580.335,Z 467.316,A -85,B 0,C 180,E1 -1707.224,E2 -1707.224} C_VEL
LIN {X 0,Y 580.351,Z 467.324,A -85,B 0,C 180,E1 -1710,E2 -1710} C_VEL
LIN {X 0,Y 580.335,Z 467.316,A -85,B 0,C 180,E1 -1712.776,E2 -1712.776} C_VEL
LIN {X 0,Y 580.321,Z 467.32,A -85,B 0,C 180,E1 -1715.56,E2 -1715.56} C_VEL
LIN {X 0,Y 580.325,Z 467.322,A -85,B 0,C 180,E1 -1718.356,E2 -1718.356} C_VEL
LIN {X 0,Y 580.296,Z 467.32,A -85,B 0,C 180,E1 -1721.191,E2 -1721.191} C_VEL
LIN {X 0,Y 580.323,Z 467.327,A -85,B 0,C 180,E1 -1724.017,E2 -1724.017} C_VEL
LIN {X 0,Y 580.308,Z 467.319,A -85,B 0,C 180,E1 -1726.914,E2 -1726.914} C_VEL
LIN {X 0,Y 580.301,Z 467.325,A -85,B 0,C 180,E1 -1729.822,E2 -1729.822} C_VEL
LIN {X 0,Y 580.29,Z 467.322,A -85,B 0,C 180,E1 -1732.802,E2 -1732.802} C_VEL
LIN {X 0,Y 580.302,Z 467.32,A -85,B 0,C 180,E1 -1735.079,E2 -1735.079} C_VEL
LIN {X 0,Y 580.296,Z 467.33,A -85,B 0,C 180,E1 -1738.185,E2 -1738.185} C_VEL
LIN {X 0,Y 580.294,Z 467.323,A -85,B 0,C 180,E1 -1740.697,E2 -1740.697} C_VEL
LIN {X 0,Y 580.298,Z 467.32,A -85,B 0,C 180,E1 -1743.316,E2 -1743.316} C_VEL
LIN {X 0,Y 580.318,Z 467.32,A -85,B 0,C 180,E1 -1745.767,E2 -1745.767} C_VEL
LIN {X 0,Y 580.283,Z 467.329,A -85,B 0,C 180,E1 -1748.146,E2 -1748.146} C_VEL
LIN {X 0,Y 580.298,Z 467.32,A -85,B 0,C 180,E1 -1750.842,E2 -1750.842} C_VEL
LIN {X 0,Y 580.283,Z 467.318,A -85,B 0,C 180,E1 -1753.656,E2 -1753.656} C_VEL
LIN {X 0,Y 580.276,Z 467.327,A -85,B 0,C 180,E1 -1756.608,E2 -1756.608} C_VEL
LIN {X 0,Y 580.292,Z 467.319,A -85,B 0,C 180,E1 -1759.157,E2 -1759.157} C_VEL
LIN {X 0,Y 580.282,Z 467.326,A -85,B 0,C 180,E1 -1761.926,E2 -1761.926} C_VEL
LIN {X 0,Y 580.3,Z 467.327,A -85,B 0,C 180,E1 -1764.457,E2 -1764.457} C_VEL
LIN {X 0,Y 580.283,Z 467.322,A -85,B 0,C 180,E1 -1766.975,E2 -1766.975} C_VEL
LIN {X 0,Y 580.3,Z 467.317,A -85,B 0,C 180,E1 -1769.426,E2 -1769.426} C_VEL
LIN {X 0,Y 580.31,Z 467.325,A -85,B 0,C 180,E1 -1772.137,E2 -1772.137} C_VEL
LIN {X 0,Y 580.3,Z 467.319,A -85,B 0,C 180,E1 -1774.92,E2 -1774.92} C_VEL
LIN {X 0,Y 580.265,Z 467.327,A -85,B 0,C 180,E1 -1777.948,E2 -1777.948} C_VEL
LIN {X 0,Y 580.307,Z 467.319,A -85,B 0,C 180,E1 -1780.914,E2 -1780.914} C_VEL
LIN {X 0,Y 580.273,Z 467.323,A -85,B 0,C 180,E1 -1783.826,E2 -1783.826} C_VEL
LIN {X 0,Y 580.315,Z 467.321,A -85,B 0,C 180,E1 -1785.983,E2 -1785.983} C_VEL
LIN {X 0,Y 580.321,Z 467.318,A -85,B 0,C 180,E1 -1788.828,E2 -1788.828} C_VEL
LIN {X 0,Y 580.327,Z 467.315,A -85,B 0,C 180,E1 -1791.644,E2 -1791.644} C_VEL
LIN {X 0,Y 580.317,Z 467.327,A -85,B 0,C 180,E1 -1794.441,E2 -1794.441} C_VEL
LIN {X 0,Y 580.339,Z 467.312,A -85,B 0,C 180,E1 -1797.224,E2 -1797.224} C_VEL
LIN {X 0,Y 580.342,Z 467.315,A -85,B 0,C 180,E1 -1800,E2 -1800} C_VEL
LIN {X 0,Y 580.339,Z 467.319,A -85,B 0,C 180,E1 -1802.777,E2 -1802.777} C_VEL
LIN {X 0,Y 580.317,Z 467.314,A -85,B 0,C 180,E1 -1805.56,E2 -1805.56} C_VEL
LIN {X 0,Y 580.327,Z 467.322,A -85,B 0,C 180,E1 -1808.356,E2 -1808.356} C_VEL
LIN {X 0,Y 580.289,Z 467.321,A -85,B 0,C 180,E1 -1811.192,E2 -1811.192} C_VEL
LIN {X 0,Y 580.316,Z 467.316,A -85,B 0,C 180,E1 -1814.017,E2 -1814.017} C_VEL
LIN {X 0,Y 580.304,Z 467.324,A -85,B 0,C 180,E1 -1816.915,E2 -1816.915} C_VEL
LIN {X 0,Y 580.299,Z 467.318,A -85,B 0,C 180,E1 -1819.823,E2 -1819.823} C_VEL
LIN {X 0,Y 580.266,Z 467.324,A -85,B 0,C 180,E1 -1822.053,E2 -1822.053} C_VEL
LIN {X 0,Y 580.302,Z 467.322,A -85,B 0,C 180,E1 -1825.08,E2 -1825.08} C_VEL
LIN {X 0,Y 580.313,Z 467.316,A -85,B 0,C 180,E1 -1827.864,E2 -1827.864} C_VEL
LIN {X 0,Y 580.286,Z 467.331,A -85,B 0,C 180,E1 -1830.697,E2 -1830.697} C_VEL
LIN {X 0,Y 580.298,Z 467.32,A -85,B 0,C 180,E1 -1833.317,E2 -1833.317} C_VEL
LIN {X 0,Y 580.321,Z 467.317,A -85,B 0,C 180,E1 -1835.768,E2 -1835.768} C_VEL
LIN {X 0,Y 580.283,Z 467.322,A -85,B 0,C 180,E1 -1838.147,E2 -1838.147} C_VEL
LIN {X 0,Y 580.294,Z 467.328,A -85,B 0,C 180,E1 -1840.844,E2 -1840.844} C_VEL
LIN {X 0,Y 580.273,Z 467.323,A -85,B 0,C 180,E1 -1843.659,E2 -1843.659} C_VEL
LIN {X 0,Y 580.282,Z 467.328,A -85,B 0,C 180,E1 -1846.609,E2 -1846.609} C_VEL
LIN {X 0,Y 580.297,Z 467.324,A -85,B 0,C 180,E1 -1849.158,E2 -1849.158} C_VEL
LIN {X 0,Y 580.289,Z 467.318,A -85,B 0,C 180,E1 -1851.928,E2 -1851.928} C_VEL
LIN {X 0,Y 580.248,Z 467.324,A -85,B 0,C 180,E1 -1854.453,E2 -1854.453} C_VEL
LIN {X 0,Y 580.289,Z 467.328,A -85,B 0,C 180,E1 -1856.976,E2 -1856.976} C_VEL
LIN {X 0,Y 580.302,Z 467.32,A -85,B 0,C 180,E1 -1859.426,E2 -1859.426} C_VEL
LIN {X 0,Y 580.297,Z 467.321,A -85,B 0,C 180,E1 -1862.142,E2 -1862.142} C_VEL
LIN {X 0,Y 580.345,Z 467.54,A -85,B 0,C 180,E1 -1864.08,E2 -1864.08} C_VEL
LIN {X 0,Y 581.02,Z 472.564,A -85,B 0,C 180,E1 -1864.954,E2 -1864.954} C_VEL
LIN {X 0,Y 580.829,Z 491.17,A -85,B 0,C 180,E1 -1867.97,E2 -1867.97} C_VEL
LIN {X 0,Y 580.621,Z 509.777,A -85,B 0,C 180,E1 -1870.925,E2 -1870.925} C_VEL
LIN {X 0,Y 580.528,Z 525.91,A -85,B 0,C 180,E1 -1873.426,E2 -1873.426} C_VEL
LIN {X 0,Y 581.043,Z 528.991,A -85,B 0,C 180,E1 -1873.514,E2 -1873.514} C_VEL
LIN {X 0,Y 581.427,Z 532.223,A -85,B 0,C 180,E1 -1873.566,E2 -1873.566} C_VEL
LIN {X 0,Y 581.158,Z 661.426,A -85,B 0,C 180,E1 -1875.199,E2 -1875.199} C_VEL
LIN {X 0,Y 581.071,Z 674.832,A -85,B 0,C 180,E1 -1875.485,E2 -1875.485} C_VEL
LIN {X 0,Y 580.963,Z 689.239,A -85,B 0,C 180,E1 -1875.94,E2 -1875.94} C_VEL
LIN {X 0,Y 580.841,Z 702.834,A -85,B 0,C 180,E1 -1876.531,E2 -1876.531} C_VEL
LIN {X 0,Y 580.698,Z 714.215,A -85,B 0,C 180,E1 -1877.151,E2 -1877.151} C_VEL
LIN {X 0,Y 580.589,Z 726.151,A -85,B 0,C 180,E1 -1877.948,E2 -1877.948} C_VEL
LIN {X 0,Y 580.442,Z 737.011,A -85,B 0,C 180,E1 -1878.83,E2 -1878.83} C_VEL
LIN {X 0,Y 580.324,Z 747.718,A -85,B 0,C 180,E1 -1879.887,E2 -1879.887} C_VEL
LIN {X 0,Y 580.277,Z 756.548,A -85,B 0,C 180,E1 -1880.941,E2 -1880.941} C_VEL
LIN {X 0,Y 580.188,Z 763.902,A -85,B 0,C 180,E1 -1881.993,E2 -1881.993} C_VEL
LIN {X 0,Y 580.141,Z 770.053,A -85,B 0,C 180,E1 -1883.042,E2 -1883.042} C_VEL
LIN {X 0,Y 580.128,Z 776.58,A -85,B 0,C 180,E1 -1884.438,E2 -1884.438} C_VEL
LIN {X 0,Y 580.102,Z 781.45,A -85,B 0,C 180,E1 -1885.832,E2 -1885.832} C_VEL
LIN {X 0,Y 580.041,Z 784.815,A -85,B 0,C 180,E1 -1887.222,E2 -1887.222} C_VEL
LIN {X 0,Y 580.041,Z 786.817,A -85,B 0,C 180,E1 -1888.611,E2 -1888.611} C_VEL
LIN {X 0,Y 580.036,Z 787.5,A -85,B 0,C 180,E1 -1890,E2 -1890} C_VEL
LIN {X 0,Y 580.041,Z 786.817,A -85,B 0,C 180,E1 -1891.389,E2 -1891.389} C_VEL
LIN {X 0,Y 580.041,Z 784.815,A -85,B 0,C 180,E1 -1892.778,E2 -1892.778} C_VEL
LIN {X 0,Y 580.102,Z 781.45,A -85,B 0,C 180,E1 -1894.168,E2 -1894.168} C_VEL
LIN {X 0,Y 580.128,Z 776.58,A -85,B 0,C 180,E1 -1895.562,E2 -1895.562} C_VEL
LIN {X 0,Y 580.141,Z 770.053,A -85,B 0,C 180,E1 -1896.958,E2 -1896.958} C_VEL
LIN {X 0,Y 580.192,Z 762.774,A -85,B 0,C 180,E1 -1898.183,E2 -1898.183} C_VEL
LIN {X 0,Y 580.284,Z 753.826,A -85,B 0,C 180,E1 -1899.41,E2 -1899.41} C_VEL
LIN {X 0,Y 580.356,Z 744.382,A -85,B 0,C 180,E1 -1900.465,E2 -1900.465} C_VEL
LIN {X 0,Y 580.469,Z 734.28,A -85,B 0,C 180,E1 -1901.404,E2 -1901.404} C_VEL
LIN {X 0,Y 580.582,Z 723.678,A -85,B 0,C 180,E1 -1902.23,E2 -1902.23} C_VEL
LIN {X 0,Y 580.701,Z 711.237,A -85,B 0,C 180,E1 -1903.027,E2 -1903.027} C_VEL
LIN {X 0,Y 580.904,Z 697.192,A -85,B 0,C 180,E1 -1903.735,E2 -1903.735} C_VEL
LIN {X 0,Y 581.017,Z 684.158,A -85,B 0,C 180,E1 -1904.236,E2 -1904.236} C_VEL
LIN {X 0,Y 581.059,Z 671.829,A -85,B 0,C 180,E1 -1904.589,E2 -1904.589} C_VEL
LIN {X 0,Y 581.195,Z 658.651,A -85,B 0,C 180,E1 -1904.845,E2 -1904.845} C_VEL
LIN {X 0,Y 581.328,Z 530.435,A -85,B 0,C 180,E1 -1906.46,E2 -1906.46} C_VEL
LIN {X 0,Y 580.556,Z 526.244,A -85,B 0,C 180,E1 -1906.55,E2 -1906.55} C_VEL
LIN {X 0,Y 580.495,Z 523.214,A -85,B 0,C 180,E1 -1906.972,E2 -1906.972} C_VEL
LIN {X 0,Y 580.647,Z 505.125,A -85,B 0,C 180,E1 -1909.81,E2 -1909.81} C_VEL
LIN {X 0,Y 580.86,Z 487.682,A -85,B 0,C 180,E1 -1912.591,E2 -1912.591} C_VEL
LIN {X 0,Y 580.989,Z 471.401,A -85,B 0,C 180,E1 -1915.239,E2 -1915.239} C_VEL
LIN {X 0,Y 580.339,Z 467.43,A -85,B 0,C 180,E1 -1915.958,E2 -1915.958} C_VEL
LIN {X 0,Y 580.291,Z 467.328,A -85,B 0,C 180,E1 -1918.975,E2 -1918.975} C_VEL
LIN {X 0,Y 580.287,Z 467.327,A -85,B 0,C 180,E1 -1921.384,E2 -1921.384} C_VEL
LIN {X 0,Y 580.314,Z 467.319,A -85,B 0,C 180,E1 -1923.854,E2 -1923.854} C_VEL
LIN {X 0,Y 580.296,Z 467.318,A -85,B 0,C 180,E1 -1926.934,E2 -1926.934} C_VEL
LIN {X 0,Y 580.291,Z 467.322,A -85,B 0,C 180,E1 -1929.932,E2 -1929.932} C_VEL
LIN {X 0,Y 580.279,Z 467.323,A -85,B 0,C 180,E1 -1932.705,E2 -1932.705} C_VEL
LIN {X 0,Y 580.265,Z 467.328,A -85,B 0,C 180,E1 -1935.608,E2 -1935.608} C_VEL
LIN {X 0,Y 580.284,Z 467.32,A -85,B 0,C 180,E1 -1938.231,E2 -1938.231} C_VEL
LIN {X 0,Y 580.284,Z 467.326,A -85,B 0,C 180,E1 -1940.965,E2 -1940.965} C_VEL
LIN {X 0,Y 580.291,Z 467.326,A -85,B 0,C 180,E1 -1943.598,E2 -1943.598} C_VEL
LIN {X 0,Y 580.314,Z 467.316,A -85,B 0,C 180,E1 -1946.145,E2 -1946.145} C_VEL
LIN {X 0,Y 580.281,Z 467.322,A -85,B 0,C 180,E1 -1948.615,E2 -1948.615} C_VEL
LIN {X 0,Y 580.289,Z 467.326,A -85,B 0,C 180,E1 -1951.023,E2 -1951.023} C_VEL
LIN {X 0,Y 580.321,Z 467.321,A -85,B 0,C 180,E1 -1953.658,E2 -1953.658} C_VEL
LIN {X 0,Y 580.272,Z 467.323,A -85,B 0,C 180,E1 -1956.441,E2 -1956.441} C_VEL
LIN {X 0,Y 580.275,Z 467.33,A -85,B 0,C 180,E1 -1959.437,E2 -1959.437} C_VEL
LIN {X 0,Y 580.275,Z 467.329,A -85,B 0,C 180,E1 -1961.645,E2 -1961.645} C_VEL
LIN {X 0,Y 580.274,Z 467.326,A -85,B 0,C 180,E1 -1963.825,E2 -1963.825} C_VEL
LIN {X 0,Y 580.316,Z 467.316,A -85,B 0,C 180,E1 -1965.983,E2 -1965.983} C_VEL
LIN {X 0,Y 580.294,Z 467.321,A -85,B 0,C 180,E1 -1968.826,E2 -1968.826} C_VEL
LIN {X 0,Y 580.327,Z 467.322,A -85,B 0,C 180,E1 -1971.644,E2 -1971.644} C_VEL
LIN {X 0,Y 580.317,Z 467.314,A -85,B 0,C 180,E1 -1974.44,E2 -1974.44} C_VEL
LIN {X 0,Y 580.339,Z 467.319,A -85,B 0,C 180,E1 -1977.223,E2 -1977.223} C_VEL
LIN {X 0,Y 580.342,Z 467.315,A -85,B 0,C 180,E1 -1980,E2 -1980} C_VEL
LIN {X 0,Y 580.339,Z 467.312,A -85,B 0,C 180,E1 -1982.776,E2 -1982.776} C_VEL
LIN {X 0,Y 580.315,Z 467.328,A -85,B 0,C 180,E1 -1985.559,E2 -1985.559} C_VEL
LIN {X 0,Y 580.327,Z 467.315,A -85,B 0,C 180,E1 -1988.356,E2 -1988.356} C_VEL
LIN {X 0,Y 580.323,Z 467.319,A -85,B 0,C 180,E1 -1991.208,E2 -1991.208} C_VEL
LIN {X 0,Y 580.304,Z 467.319,A -85,B 0,C 180,E1 -1994.339,E2 -1994.339} C_VEL
LIN {X 0,Y 580.303,Z 467.318,A -85,B 0,C 180,E1 -1996.915,E2 -1996.915} C_VEL
LIN {X 0,Y 580.298,Z 467.326,A -85,B 0,C 180,E1 -1999.822,E2 -1999.822} C_VEL
LIN {X 0,Y 580.277,Z 467.327,A -85,B 0,C 180,E1 -2001.344,E2 -2001.344} C_VEL
LIN {X 0,Y 579.579,Z 467.414,A -85,B 0,C 180,E1 -2001.924,E2 -2001.924} C_VEL
LIN {X 0,Y 576.701,Z 467.768,A -85,B 0,C 180,E1 -2002.863,E2 -2002.863} C_VEL
LIN {X 0,Y 574.306,Z 468.074,A -85,B 0,C 180,E1 -2003.62,E2 -2003.62} C_VEL
LIN {X 0,Y 573.308,Z 468.19,A -85,B 0,C 180,E1 -2004.203,E2 -2004.203} C_VEL
LIN {X 0,Y 573.241,Z 468.197,A -85,B 0,C 180,E1 -2004.401,E2 -2004.401} C_VEL
LIN {X 0,Y 573.255,Z 468.198,A -85,B 0,C 180,E1 -2006.975,E2 -2006.975} C_VEL
LIN {X 0,Y 573.245,Z 468.205,A -85,B 0,C 180,E1 -2009.49,E2 -2009.49} C_VEL
LIN {X 0,Y 573.247,Z 468.2,A -85,B 0,C 180,E1 -2012.229,E2 -2012.229} C_VEL
LIN {X 0,Y 573.245,Z 468.198,A -85,B 0,C 180,E1 -2014.775,E2 -2014.775} C_VEL
LIN {X 0,Y 573.244,Z 468.199,A -85,B 0,C 180,E1 -2017.166,E2 -2017.166} C_VEL
LIN {X 0,Y 573.241,Z 468.207,A -85,B 0,C 180,E1 -2019.607,E2 -2019.607} C_VEL
LIN {X 0,Y 573.234,Z 468.2,A -85,B 0,C 180,E1 -2022.642,E2 -2022.642} C_VEL
LIN {X 0,Y 573.231,Z 468.207,A -85,B 0,C 180,E1 -2025.667,E2 -2025.667} C_VEL
LIN {X 0,Y 573.253,Z 468.197,A -85,B 0,C 180,E1 -2028.546,E2 -2028.546} C_VEL
LIN {X 0,Y 573.243,Z 468.202,A -85,B 0,C 180,E1 -2031.3,E2 -2031.3} C_VEL
LIN {X 0,Y 573.257,Z 468.203,A -85,B 0,C 180,E1 -2034.012,E2 -2034.012} C_VEL
LIN {X 0,Y 573.278,Z 468.195,A -85,B 0,C 180,E1 -2036.519,E2 -2036.519} C_VEL
LIN {X 0,Y 573.238,Z 468.2,A -85,B 0,C 180,E1 -2039.115,E2 -2039.115} C_VEL
LIN {X 0,Y 573.258,Z 468.206,A -85,B 0,C 180,E1 -2041.969,E2 -2041.969} C_VEL
LIN {X 0,Y 573.249,Z 468.199,A -85,B 0,C 180,E1 -2044.59,E2 -2044.59} C_VEL
LIN {X 0,Y 573.233,Z 468.207,A -85,B 0,C 180,E1 -2047.663,E2 -2047.663} C_VEL
LIN {X 0,Y 573.274,Z 468.196,A -85,B 0,C 180,E1 -2050.729,E2 -2050.729} C_VEL
LIN {X 0,Y 573.249,Z 468.204,A -85,B 0,C 180,E1 -2053.622,E2 -2053.622} C_VEL
LIN {X 0,Y 573.27,Z 468.204,A -85,B 0,C 180,E1 -2055.807,E2 -2055.807} C_VEL
LIN {X 0,Y 573.259,Z 468.198,A -85,B 0,C 180,E1 -2058.745,E2 -2058.745} C_VEL
LIN {X 0,Y 573.281,Z 468.198,A -85,B 0,C 180,E1 -2061.541,E2 -2061.541} C_VEL
LIN {X 0,Y 573.287,Z 468.198,A -85,B 0,C 180,E1 -2064.372,E2 -2064.372} C_VEL
LIN {X 0,Y 573.311,Z 468.2,A -85,B 0,C 180,E1 -2067.892,E2 -2067.892} C_VEL
LIN {X 0,Y 573.327,Z 468.19,A -85,B 0,C 180,E1 -2070.702,E2 -2070.702} C_VEL
LIN {X 0,Y 573.302,Z 468.193,A -85,B 0,C 180,E1 -2072.811,E2 -2072.811} C_VEL
LIN {X 0,Y 573.288,Z 468.198,A -85,B 0,C 180,E1 -2075.628,E2 -2075.628} C_VEL
LIN {X 0,Y 573.281,Z 468.198,A -85,B 0,C 180,E1 -2078.459,E2 -2078.459} C_VEL
LIN {X 0,Y 573.268,Z 468.197,A -85,B 0,C 180,E1 -2081.312,E2 -2081.312} C_VEL
LIN {X 0,Y 573.278,Z 468.2,A -85,B 0,C 180,E1 -2084.424,E2 -2084.424} C_VEL
LIN {X 0,Y 573.255,Z 468.198,A -85,B 0,C 180,E1 -2087.111,E2 -2087.111} C_VEL
LIN {X 0,Y 573.248,Z 468.208,A -85,B 0,C 180,E1 -2090.076,E2 -2090.076} C_VEL
LIN {X 0,Y 573.229,Z 468.201,A -85,B 0,C 180,E1 -2093.099,E2 -2093.099} C_VEL
LIN {X 0,Y 573.249,Z 468.199,A -85,B 0,C 180,E1 -2095.41,E2 -2095.41} C_VEL
LIN {X 0,Y 573.258,Z 468.206,A -85,B 0,C 180,E1 -2098.031,E2 -2098.031} C_VEL
LIN {X 0,Y 573.238,Z 468.2,A -85,B 0,C 180,E1 -2100.885,E2 -2100.885} C_VEL
LIN {X 0,Y 573.255,Z 468.199,A -85,B 0,C 180,E1 -2103.524,E2 -2103.524} C_VEL
LIN {X 0,Y 573.254,Z 468.205,A -85,B 0,C 180,E1 -2106.048,E2 -2106.048} C_VEL
LIN {X 0,Y 573.243,Z 468.202,A -85,B 0,C 180,E1 -2108.7,E2 -2108.7} C_VEL
LIN {X 0,Y 573.247,Z 468.198,A -85,B 0,C 180,E1 -2111.596,E2 -2111.596} C_VEL
LIN {X 0,Y 573.231,Z 468.207,A -85,B 0,C 180,E1 -2114.333,E2 -2114.333} C_VEL
LIN {X 0,Y 573.234,Z 468.2,A -85,B 0,C 180,E1 -2117.358,E2 -2117.358} C_VEL
LIN {X 0,Y 573.241,Z 468.207,A -85,B 0,C 180,E1 -2120.393,E2 -2120.393} C_VEL
LIN {X 0,Y 573.247,Z 468.197,A -85,B 0,C 180,E1 -2123.078,E2 -2123.078} C_VEL
LIN {X 0,Y 573.266,Z 468.196,A -85,B 0,C 180,E1 -2125.672,E2 -2125.672} C_VEL
LIN {X 0,Y 573.241,Z 468.207,A -85,B 0,C 180,E1 -2128.185,E2 -2128.185} C_VEL
LIN {X 0,Y 573.261,Z 468.201,A -85,B 0,C 180,E1 -2130.634,E2 -2130.634} C_VEL
LIN {X 0,Y 573.261,Z 468.196,A -85,B 0,C 180,E1 -2133.5,E2 -2133.5} C_VEL
LIN {X 0,Y 573.223,Z 468.205,A -85,B 0,C 180,E1 -2136.135,E2 -2136.135} C_VEL
LIN {X 0,Y 573.251,Z 468.198,A -85,B 0,C 180,E1 -2139.174,E2 -2139.174} C_VEL
LIN {X 0,Y 573.229,Z 468.198,A -85,B 0,C 180,E1 -2141.412,E2 -2141.412} C_VEL
LIN {X 0,Y 573.249,Z 468.196,A -85,B 0,C 180,E1 -2143.622,E2 -2143.622} C_VEL
LIN {X 0,Y 573.228,Z 468.209,A -85,B 0,C 180,E1 -2146.53,E2 -2146.53} C_VEL
LIN {X 0,Y 573.273,Z 468.197,A -85,B 0,C 180,E1 -2148.734,E2 -2148.734} C_VEL
LIN {X 0,Y 573.298,Z 468.19,A -85,B 0,C 180,E1 -2151.541,E2 -2151.541} C_VEL
LIN {X 0,Y 573.283,Z 468.202,A -85,B 0,C 180,E1 -2154.372,E2 -2154.372} C_VEL
LIN {X 0,Y 573.3,Z 468.189,A -85,B 0,C 180,E1 -2157.893,E2 -2157.893} C_VEL
LIN {X 0,Y 573.328,Z 468.194,A -85,B 0,C 180,E1 -2160.703,E2 -2160.703} C_VEL
LIN {X 0,Y 573.232,Z 468.199,A -85,B 0,C 180,E1 -2163.515,E2 -2163.515} C_VEL
LIN {X 0,Y 573.284,Z 468.189,A -85,B 0,C 180,E1 -2165.629,E2 -2165.629} C_VEL
LIN {X 0,Y 573.298,Z 468.199,A -85,B 0,C 180,E1 -2168.46,E2 -2168.46} C_VEL
LIN {X 0,Y 573.261,Z 468.196,A -85,B 0,C 180,E1 -2171.312,E2 -2171.312} C_VEL
LIN {X 0,Y 573.263,Z 468.196,A -85,B 0,C 180,E1 -2174.194,E2 -2174.194} C_VEL
LIN {X 0,Y 573.251,Z 468.2,A -85,B 0,C 180,E1 -2177.112,E2 -2177.112} C_VEL
LIN {X 0,Y 573.248,Z 468.198,A -85,B 0,C 180,E1 -2180.077,E2 -2180.077} C_VEL
LIN {X 0,Y 573.23,Z 468.204,A -85,B 0,C 180,E1 -2182.338,E2 -2182.338} C_VEL
LIN {X 0,Y 573.25,Z 468.197,A -85,B 0,C 180,E1 -2185.411,E2 -2185.411} C_VEL
LIN {X 0,Y 573.257,Z 468.196,A -85,B 0,C 180,E1 -2188.032,E2 -2188.032} C_VEL
LIN {X 0,Y 573.232,Z 468.206,A -85,B 0,C 180,E1 -2190.885,E2 -2190.885} C_VEL
LIN {X 0,Y 573.255,Z 468.196,A -85,B 0,C 180,E1 -2193.525,E2 -2193.525} C_VEL
LIN {X 0,Y 573.255,Z 468.198,A -85,B 0,C 180,E1 -2196.049,E2 -2196.049} C_VEL
LIN {X 0,Y 573.243,Z 468.207,A -85,B 0,C 180,E1 -2198.702,E2 -2198.702} C_VEL
LIN {X 0,Y 573.23,Z 468.2,A -85,B 0,C 180,E1 -2201.457,E2 -2201.457} C_VEL
LIN {X 0,Y 573.23,Z 468.204,A -85,B 0,C 180,E1 -2204.334,E2 -2204.334} C_VEL
LIN {X 0,Y 573.24,Z 468.199,A -85,B 0,C 180,E1 -2207.359,E2 -2207.359} C_VEL
LIN {X 0,Y 573.244,Z 468.203,A -85,B 0,C 180,E1 -2210.394,E2 -2210.394} C_VEL
LIN {X 0,Y 573.25,Z 468.194,A -85,B 0,C 180,E1 -2213.078,E2 -2213.078} C_VEL
LIN {X 0,Y 573.265,Z 468.197,A -85,B 0,C 180,E1 -2215.672,E2 -2215.672} C_VEL
LIN {X 0,Y 573.247,Z 468.199,A -85,B 0,C 180,E1 -2218.186,E2 -2218.186} C_VEL
LIN {X 0,Y 573.263,Z 468.203,A -85,B 0,C 180,E1 -2220.635,E2 -2220.635} C_VEL
LIN {X 0,Y 573.25,Z 468.198,A -85,B 0,C 180,E1 -2223.025,E2 -2223.025} C_VEL
LIN {X 0,Y 573.306,Z 468.329,A -85,B 0,C 180,E1 -2223.862,E2 -2223.862} C_VEL
LIN {X 0,Y 574.086,Z 472.564,A -85,B 0,C 180,E1 -2224.63,E2 -2224.63} C_VEL
LIN {X 0,Y 573.916,Z 488.845,A -85,B 0,C 180,E1 -2227.311,E2 -2227.311} C_VEL
LIN {X 0,Y 573.679,Z 505.125,A -85,B 0,C 180,E1 -2229.939,E2 -2229.939} C_VEL
LIN {X 0,Y 573.564,Z 522.568,A -85,B 0,C 180,E1 -2232.714,E2 -2232.714} C_VEL
LIN {X 0,Y 573.571,Z 526.198,A -85,B 0,C 180,E1 -2233.24,E2 -2233.24} C_VEL
LIN {X 0,Y 574.572,Z 531.654,A -85,B 0,C 180,E1 -2233.357,E2 -2233.357} C_VEL
LIN {X 0,Y 574.31,Z 661.378,A -85,B 0,C 180,E1 -2235.019,E2 -2235.019} C_VEL
LIN {X 0,Y 574.19,Z 674.19,A -85,B 0,C 180,E1 -2235.292,E2 -2235.292} C_VEL
LIN {X 0,Y 574.086,Z 687.839,A -85,B 0,C 180,E1 -2235.716,E2 -2235.716} C_VEL
LIN {X 0,Y 573.927,Z 701.073,A -85,B 0,C 180,E1 -2236.276,E2 -2236.276} C_VEL
LIN {X 0,Y 573.74,Z 712.74,A -85,B 0,C 180,E1 -2236.902,E2 -2236.902} C_VEL
LIN {X 0,Y 573.602,Z 723.665,A -85,B 0,C 180,E1 -2237.619,E2 -2237.619} C_VEL
LIN {X 0,Y 573.49,Z 733.906,A -85,B 0,C 180,E1 -2238.424,E2 -2238.424} C_VEL
LIN {X 0,Y 573.354,Z 744.38,A -85,B 0,C 180,E1 -2239.405,E2 -2239.405} C_VEL
LIN {X 0,Y 573.253,Z 753.826,A -85,B 0,C 180,E1 -2240.473,E2 -2240.473} C_VEL
LIN {X 0,Y 573.151,Z 761.637,A -85,B 0,C 180,E1 -2241.539,E2 -2241.539} C_VEL
LIN {X 0,Y 573.089,Z 768.145,A -85,B 0,C 180,E1 -2242.602,E2 -2242.602} C_VEL
LIN {X 0,Y 573.018,Z 773.522,A -85,B 0,C 180,E1 -2243.663,E2 -2243.663} C_VEL
LIN {X 0,Y 573.001,Z 777.932,A -85,B 0,C 180,E1 -2244.722,E2 -2244.722} C_VEL
LIN {X 0,Y 573.028,Z 781.451,A -85,B 0,C 180,E1 -2245.78,E2 -2245.78} C_VEL
LIN {X 0,Y 572.956,Z 784.809,A -85,B 0,C 180,E1 -2247.188,E2 -2247.188} C_VEL
LIN {X 0,Y 572.94,Z 786.814,A -85,B 0,C 180,E1 -2248.594,E2 -2248.594} C_VEL
LIN {X 0,Y 572.937,Z 787.5,A -85,B 0,C 180,E1 -2250,E2 -2250} C_VEL
LIN {X 0,Y 572.94,Z 786.814,A -85,B 0,C 180,E1 -2251.406,E2 -2251.406} C_VEL
LIN {X 0,Y 572.956,Z 784.809,A -85,B 0,C 180,E1 -2252.812,E2 -2252.812} C_VEL
LIN {X 0,Y 573.028,Z 781.451,A -85,B 0,C 180,E1 -2254.22,E2 -2254.22} C_VEL
LIN {X 0,Y 573.055,Z 776.583,A -85,B 0,C 180,E1 -2255.63,E2 -2255.63} C_VEL
LIN {X 0,Y 573.058,Z 771.86,A -85,B 0,C 180,E1 -2256.693,E2 -2256.693} C_VEL
LIN {X 0,Y 573.126,Z 765.019,A -85,B 0,C 180,E1 -2257.929,E2 -2257.929} C_VEL
LIN {X 0,Y 573.197,Z 757.871,A -85,B 0,C 180,E1 -2258.994,E2 -2258.994} C_VEL
LIN {X 0,Y 573.264,Z 749.288,A -85,B 0,C 180,E1 -2260.061,E2 -2260.061} C_VEL
LIN {X 0,Y 573.45,Z 739.815,A -85,B 0,C 180,E1 -2261.046,E2 -2261.046} C_VEL
LIN {X 0,Y 573.584,Z 727.334,A -85,B 0,C 180,E1 -2262.112,E2 -2262.112} C_VEL
LIN {X 0,Y 573.746,Z 715.662,A -85,B 0,C 180,E1 -2262.917,E2 -2262.917} C_VEL
LIN {X 0,Y 573.882,Z 704.573,A -85,B 0,C 180,E1 -2263.545,E2 -2263.545} C_VEL
LIN {X 0,Y 574.044,Z 691.841,A -85,B 0,C 180,E1 -2264.128,E2 -2264.128} C_VEL
LIN {X 0,Y 574.163,Z 676.795,A -85,B 0,C 180,E1 -2264.642,E2 -2264.642} C_VEL
LIN {X 0,Y 574.28,Z 662.737,A -85,B 0,C 180,E1 -2264.96,E2 -2264.96} C_VEL
LIN {X 0,Y 574.43,Z 607.347,A -85,B 0,C 180,E1 -2265.682,E2 -2265.682} C_VEL
LIN {X 0,Y 574.55,Z 531.542,A -85,B 0,C 180,E1 -2266.645,E2 -2266.645} C_VEL
LIN {X 0,Y 573.564,Z 526.202,A -85,B 0,C 180,E1 -2266.761,E2 -2266.761} C_VEL
LIN {X 0,Y 573.564,Z 522.568,A -85,B 0,C 180,E1 -2267.286,E2 -2267.286} C_VEL
LIN {X 0,Y 573.755,Z 502.799,A -85,B 0,C 180,E1 -2270.432,E2 -2270.432} C_VEL
LIN {X 0,Y 573.945,Z 486.519,A -85,B 0,C 180,E1 -2273.069,E2 -2273.069} C_VEL
LIN {X 0,Y 574.067,Z 472.564,A -85,B 0,C 180,E1 -2275.371,E2 -2275.371} C_VEL
LIN {X 0,Y 573.28,Z 468.281,A -85,B 0,C 180,E1 -2276.164,E2 -2276.164} C_VEL
LIN {X 0,Y 573.236,Z 468.201,A -85,B 0,C 180,E1 -2278.564,E2 -2278.564} C_VEL
LIN {X 0,Y 573.235,Z 468.201,A -85,B 0,C 180,E1 -2280.992,E2 -2280.992} C_VEL
LIN {X 0,Y 573.261,Z 468.202,A -85,B 0,C 180,E1 -2283.523,E2 -2283.523} C_VEL
LIN {X 0,Y 573.212,Z 468.195,A -85,B 0,C 180,E1 -2286.051,E2 -2286.051} C_VEL
LIN {X 0,Y 573.246,Z 468.197,A -85,B 0,C 180,E1 -2288.7,E2 -2288.7} C_VEL
LIN {X 0,Y 573.25,Z 468.201,A -85,B 0,C 180,E1 -2291.595,E2 -2291.595} C_VEL
LIN {X 0,Y 573.235,Z 468.198,A -85,B 0,C 180,E1 -2294.332,E2 -2294.332} C_VEL
LIN {X 0,Y 573.235,Z 468.207,A -85,B 0,C 180,E1 -2297.358,E2 -2297.358} C_VEL
LIN {X 0,Y 573.243,Z 468.199,A -85,B 0,C 180,E1 -2300.392,E2 -2300.392} C_VEL
LIN {X 0,Y 573.25,Z 468.203,A -85,B 0,C 180,E1 -2303.077,E2 -2303.077} C_VEL
LIN {X 0,Y 573.269,Z 468.198,A -85,B 0,C 180,E1 -2305.671,E2 -2305.671} C_VEL
LIN {X 0,Y 573.242,Z 468.198,A -85,B 0,C 180,E1 -2308.184,E2 -2308.184} C_VEL
LIN {X 0,Y 573.26,Z 468.197,A -85,B 0,C 180,E1 -2310.634,E2 -2310.634} C_VEL
LIN {X 0,Y 573.263,Z 468.203,A -85,B 0,C 180,E1 -2313.5,E2 -2313.5} C_VEL
LIN {X 0,Y 573.225,Z 468.201,A -85,B 0,C 180,E1 -2316.134,E2 -2316.134} C_VEL
LIN {X 0,Y 573.254,Z 468.202,A -85,B 0,C 180,E1 -2319.173,E2 -2319.173} C_VEL
LIN {X 0,Y 573.232,Z 468.209,A -85,B 0,C 180,E1 -2321.411,E2 -2321.411} C_VEL
LIN {X 0,Y 573.25,Z 468.204,A -85,B 0,C 180,E1 -2323.621,E2 -2323.621} C_VEL
LIN {X 0,Y 573.227,Z 468.197,A -85,B 0,C 180,E1 -2326.529,E2 -2326.529} C_VEL
LIN {X 0,Y 573.252,Z 468.197,A -85,B 0,C 180,E1 -2328.744,E2 -2328.744} C_VEL
LIN {X 0,Y 573.298,Z 468.199,A -85,B 0,C 180,E1 -2331.54,E2 -2331.54} C_VEL
LIN {X 0,Y 573.284,Z 468.189,A -85,B 0,C 180,E1 -2334.371,E2 -2334.371} C_VEL
LIN {X 0,Y 573.3,Z 468.195,A -85,B 0,C 180,E1 -2337.892,E2 -2337.892} C_VEL
LIN {X 0,Y 573.328,Z 468.186,A -85,B 0,C 180,E1 -2340.702,E2 -2340.702} C_VEL
LIN {X 0,Y 573.233,Z 468.207,A -85,B 0,C 180,E1 -2343.514,E2 -2343.514} C_VEL
LIN {X 0,Y 573.282,Z 468.202,A -85,B 0,C 180,E1 -2345.628,E2 -2345.628} C_VEL
LIN {X 0,Y 573.298,Z 468.19,A -85,B 0,C 180,E1 -2348.459,E2 -2348.459} C_VEL
LIN {X 0,Y 573.289,Z 468.196,A -85,B 0,C 180,E1 -2351.311,E2 -2351.311} C_VEL
LIN {X 0,Y 573.27,Z 468.195,A -85,B 0,C 180,E1 -2354.425,E2 -2354.425} C_VEL
LIN {X 0,Y 573.25,Z 468.198,A -85,B 0,C 180,E1 -2357.111,E2 -2357.111} C_VEL
LIN {X 0,Y 573.247,Z 468.201,A -85,B 0,C 180,E1 -2360.076,E2 -2360.076} C_VEL
LIN {X 0,Y 573.228,Z 468.2,A -85,B 0,C 180,E1 -2362.338,E2 -2362.338} C_VEL
LIN {X 0,Y 573.241,Z 468.197,A -85,B 0,C 180,E1 -2364.401,E2 -2364.401} C_VEL
LIN {X 0,Y 572.616,Z 468.276,A -85,B 0,C 180,E1 -2364.987,E2 -2364.987} C_VEL
LIN {X 0,Y 569.777,Z 468.635,A -85,B 0,C 180,E1 -2365.939,E2 -2365.939} C_VEL
LIN {X 0,Y 567.348,Z 468.94,A -85,B 0,C 180,E1 -2366.705,E2 -2366.705} C_VEL
LIN {X 0,Y 566.296,Z 469.069,A -85,B 0,C 180,E1 -2367.296,E2 -2367.296} C_VEL
LIN {X 0,Y 566.207,Z 469.078,A -85,B 0,C 180,E1 -2367.497,E2 -2367.497} C_VEL
LIN {X 0,Y 566.218,Z 469.079,A -85,B 0,C 180,E1 -2369.767,E2 -2369.767} C_VEL
LIN {X 0,Y 566.199,Z 469.077,A -85,B 0,C 180,E1 -2372.431,E2 -2372.431} C_VEL
LIN {X 0,Y 566.206,Z 469.075,A -85,B 0,C 180,E1 -2374.995,E2 -2374.995} C_VEL
LIN {X 0,Y 566.187,Z 469.082,A -85,B 0,C 180,E1 -2377.461,E2 -2377.461} C_VEL
LIN {X 0,Y 566.218,Z 469.075,A -85,B 0,C 180,E1 -2380.198,E2 -2380.198} C_VEL
LIN {X 0,Y 566.196,Z 469.078,A -85,B 0,C 180,E1 -2383.054,E2 -2383.054} C_VEL
LIN {X 0,Y 566.195,Z 469.074,A -85,B 0,C 180,E1 -2386.048,E2 -2386.048} C_VEL
LIN {X 0,Y 566.213,Z 469.073,A -85,B 0,C 180,E1 -2388.865,E2 -2388.865} C_VEL
LIN {X 0,Y 566.184,Z 469.086,A -85,B 0,C 180,E1 -2391.638,E2 -2391.638} C_VEL
LIN {X 0,Y 566.205,Z 469.077,A -85,B 0,C 180,E1 -2394.312,E2 -2394.312} C_VEL
LIN {X 0,Y 566.223,Z 469.074,A -85,B 0,C 180,E1 -2396.899,E2 -2396.899} C_VEL
LIN {X 0,Y 566.188,Z 469.081,A -85,B 0,C 180,E1 -2399.408,E2 -2399.408} C_VEL
LIN {X 0,Y 566.223,Z 469.083,A -85,B 0,C 180,E1 -2401.859,E2 -2401.859} C_VEL
LIN {X 0,Y 566.209,Z 469.079,A -85,B 0,C 180,E1 -2404.251,E2 -2404.251} C_VEL
LIN {X 0,Y 566.187,Z 469.078,A -85,B 0,C 180,E1 -2406.714,E2 -2406.714} C_VEL
LIN {X 0,Y 566.209,Z 469.082,A -85,B 0,C 180,E1 -2409.663,E2 -2409.663} C_VEL
LIN {X 0,Y 566.199,Z 469.078,A -85,B 0,C 180,E1 -2412.669,E2 -2412.669} C_VEL
LIN {X 0,Y 566.23,Z 469.078,A -85,B 0,C 180,E1 -2415.627,E2 -2415.627} C_VEL
LIN {X 0,Y 566.231,Z 469.074,A -85,B 0,C 180,E1 -2418.675,E2 -2418.675} C_VEL
LIN {X 0,Y 566.225,Z 469.076,A -85,B 0,C 180,E1 -2421.434,E2 -2421.434} C_VEL
LIN {X 0,Y 566.255,Z 469.075,A -85,B 0,C 180,E1 -2424.302,E2 -2424.302} C_VEL
LIN {X 0,Y 566.281,Z 469.075,A -85,B 0,C 180,E1 -2427.866,E2 -2427.866} C_VEL
LIN {X 0,Y 566.298,Z 469.066,A -85,B 0,C 180,E1 -2430.711,E2 -2430.711} C_VEL
LIN {X 0,Y 566.268,Z 469.069,A -85,B 0,C 180,E1 -2432.846,E2 -2432.846} C_VEL
LIN {X 0,Y 566.256,Z 469.075,A -85,B 0,C 180,E1 -2435.698,E2 -2435.698} C_VEL
LIN {X 0,Y 566.225,Z 469.076,A -85,B 0,C 180,E1 -2438.566,E2 -2438.566} C_VEL
LIN {X 0,Y 566.238,Z 469.074,A -85,B 0,C 180,E1 -2441.454,E2 -2441.454} C_VEL
LIN {X 0,Y 566.23,Z 469.077,A -85,B 0,C 180,E1 -2444.507,E2 -2444.507} C_VEL
LIN {X 0,Y 566.199,Z 469.078,A -85,B 0,C 180,E1 -2447.331,E2 -2447.331} C_VEL
LIN {X 0,Y 566.209,Z 469.082,A -85,B 0,C 180,E1 -2450.337,E2 -2450.337} C_VEL
LIN {X 0,Y 566.185,Z 469.079,A -85,B 0,C 180,E1 -2453.403,E2 -2453.403} C_VEL
LIN {X 0,Y 566.209,Z 469.079,A -85,B 0,C 180,E1 -2455.749,E2 -2455.749} C_VEL
LIN {X 0,Y 566.2,Z 469.086,A -85,B 0,C 180,E1 -2458.203,E2 -2458.203} C_VEL
LIN {X 0,Y 566.188,Z 469.081,A -85,B 0,C 180,E1 -2460.592,E2 -2460.592} C_VEL
LIN {X 0,Y 566.223,Z 469.074,A -85,B 0,C 180,E1 -2463.101,E2 -2463.101} C_VEL
LIN {X 0,Y 566.205,Z 469.077,A -85,B 0,C 180,E1 -2465.688,E2 -2465.688} C_VEL
LIN {X 0,Y 566.21,Z 469.079,A -85,B 0,C 180,E1 -2468.559,E2 -2468.559} C_VEL
LIN {X 0,Y 566.205,Z 469.074,A -85,B 0,C 180,E1 -2471.136,E2 -2471.136} C_VEL
LIN {X 0,Y 566.193,Z 469.076,A -85,B 0,C 180,E1 -2474.035,E2 -2474.035} C_VEL
LIN {X 0,Y 566.196,Z 469.077,A -85,B 0,C 180,E1 -2477.082,E2 -2477.082} C_VEL
LIN {X 0,Y 566.218,Z 469.075,A -85,B 0,C 180,E1 -2479.802,E2 -2479.802} C_VEL
LIN {X 0,Y 566.189,Z 469.081,A -85,B 0,C 180,E1 -2482.599,E2 -2482.599} C_VEL
LIN {X 0,Y 566.213,Z 469.074,A -85,B 0,C 180,E1 -2485.183,E2 -2485.183} C_VEL
LIN {X 0,Y 566.226,Z 469.074,A -85,B 0,C 180,E1 -2487.744,E2 -2487.744} C_VEL
LIN {X 0,Y 566.219,Z 469.081,A -85,B 0,C 180,E1 -2490.323,E2 -2490.323} C_VEL
LIN {X 0,Y 566.225,Z 469.072,A -85,B 0,C 180,E1 -2493.335,E2 -2493.335} C_VEL
LIN {X 0,Y 566.189,Z 469.076,A -85,B 0,C 180,E1 -2495.819,E2 -2495.819} C_VEL
LIN {X 0,Y 566.207,Z 469.077,A -85,B 0,C 180,E1 -2498.903,E2 -2498.903} C_VEL
LIN {X 0,Y 566.204,Z 469.074,A -85,B 0,C 180,E1 -2501.173,E2 -2501.173} C_VEL
LIN {X 0,Y 566.211,Z 469.072,A -85,B 0,C 180,E1 -2503.413,E2 -2503.413} C_VEL
LIN {X 0,Y 566.19,Z 469.086,A -85,B 0,C 180,E1 -2506.359,E2 -2506.359} C_VEL
LIN {X 0,Y 566.265,Z 469.071,A -85,B 0,C 180,E1 -2508.654,E2 -2508.654} C_VEL
LIN {X 0,Y 566.239,Z 469.069,A -85,B 0,C 180,E1 -2511.435,E2 -2511.435} C_VEL
LIN {X 0,Y 566.251,Z 469.077,A -85,B 0,C 180,E1 -2514.302,E2 -2514.302} C_VEL
LIN {X 0,Y 566.272,Z 469.064,A -85,B 0,C 180,E1 -2517.867,E2 -2517.867} C_VEL
LIN {X 0,Y 566.298,Z 469.07,A -85,B 0,C 180,E1 -2520.711,E2 -2520.711} C_VEL
LIN {X 0,Y 566.27,Z 469.071,A -85,B 0,C 180,E1 -2522.846,E2 -2522.846} C_VEL
LIN {X 0,Y 566.252,Z 469.065,A -85,B 0,C 180,E1 -2525.699,E2 -2525.699} C_VEL
LIN {X 0,Y 566.24,Z 469.081,A -85,B 0,C 180,E1 -2528.566,E2 -2528.566} C_VEL
LIN {X 0,Y 566.232,Z 469.071,A -85,B 0,C 180,E1 -2531.455,E2 -2531.455} C_VEL
LIN {X 0,Y 566.224,Z 469.078,A -85,B 0,C 180,E1 -2534.507,E2 -2534.507} C_VEL
LIN {X 0,Y 566.195,Z 469.077,A -85,B 0,C 180,E1 -2537.332,E2 -2537.332} C_VEL
LIN {X 0,Y 566.211,Z 469.078,A -85,B 0,C 180,E1 -2540.338,E2 -2540.338} C_VEL
LIN {X 0,Y 566.181,Z 469.079,A -85,B 0,C 180,E1 -2543.404,E2 -2543.404} C_VEL
LIN {X 0,Y 566.219,Z 469.073,A -85,B 0,C 180,E1 -2545.749,E2 -2545.749} C_VEL
LIN {X 0,Y 566.2,Z 469.077,A -85,B 0,C 180,E1 -2548.204,E2 -2548.204} C_VEL
LIN {X 0,Y 566.192,Z 469.08,A -85,B 0,C 180,E1 -2551.079,E2 -2551.079} C_VEL
LIN {X 0,Y 566.206,Z 469.073,A -85,B 0,C 180,E1 -2553.735,E2 -2553.735} C_VEL
LIN {X 0,Y 566.211,Z 469.083,A -85,B 0,C 180,E1 -2556.569,E2 -2556.569} C_VEL
LIN {X 0,Y 566.208,Z 469.075,A -85,B 0,C 180,E1 -2559.686,E2 -2559.686} C_VEL
LIN {X 0,Y 566.186,Z 469.078,A -85,B 0,C 180,E1 -2562.09,E2 -2562.09} C_VEL
LIN {X 0,Y 566.169,Z 469.083,A -85,B 0,C 180,E1 -2565.037,E2 -2565.037} C_VEL
LIN {X 0,Y 566.211,Z 469.073,A -85,B 0,C 180,E1 -2567.914,E2 -2567.914} C_VEL
LIN {X 0,Y 566.219,Z 469.081,A -85,B 0,C 180,E1 -2570.728,E2 -2570.728} C_VEL
LIN {X 0,Y 566.181,Z 469.069,A -85,B 0,C 180,E1 -2573.789,E2 -2573.789} C_VEL
LIN {X 0,Y 566.21,Z 469.078,A -85,B 0,C 180,E1 -2576.267,E2 -2576.267} C_VEL
LIN {X 0,Y 566.198,Z 469.077,A -85,B 0,C 180,E1 -2578.923,E2 -2578.923} C_VEL
LIN {X 0,Y 566.211,Z 469.075,A -85,B 0,C 180,E1 -2581.858,E2 -2581.858} C_VEL
LIN {X 0,Y 566.254,Z 469.297,A -85,B 0,C 180,E1 -2583.71,E2 -2583.71} C_VEL
LIN {X 0,Y 567.215,Z 475.192,A -85,B 0,C 180,E1 -2584.756,E2 -2584.756} C_VEL
LIN {X 0,Y 566.976,Z 493.496,A -85,B 0,C 180,E1 -2587.787,E2 -2587.787} C_VEL
LIN {X 0,Y 566.697,Z 510.763,A -85,B 0,C 180,E1 -2590.597,E2 -2590.597} C_VEL
LIN {X 0,Y 566.554,Z 525.926,A -85,B 0,C 180,E1 -2593.006,E2 -2593.006} C_VEL
LIN {X 0,Y 567.074,Z 528.86,A -85,B 0,C 180,E1 -2593.094,E2 -2593.094} C_VEL
LIN {X 0,Y 567.813,Z 533.542,A -85,B 0,C 180,E1 -2593.177,E2 -2593.177} C_VEL
LIN {X 0,Y 567.469,Z 661.33,A -85,B 0,C 180,E1 -2594.834,E2 -2594.834} C_VEL
LIN {X 0,Y 567.324,Z 673.477,A -85,B 0,C 180,E1 -2595.093,E2 -2595.093} C_VEL
LIN {X 0,Y 567.241,Z 686.585,A -85,B 0,C 180,E1 -2595.496,E2 -2595.496} C_VEL
LIN {X 0,Y 567.004,Z 701.062,A -85,B 0,C 180,E1 -2596.105,E2 -2596.105} C_VEL
LIN {X 0,Y 566.792,Z 712.726,A -85,B 0,C 180,E1 -2596.739,E2 -2596.739} C_VEL
LIN {X 0,Y 566.647,Z 723.653,A -85,B 0,C 180,E1 -2597.465,E2 -2597.465} C_VEL
LIN {X 0,Y 566.497,Z 733.894,A -85,B 0,C 180,E1 -2598.279,E2 -2598.279} C_VEL
LIN {X 0,Y 566.399,Z 742.929,A -85,B 0,C 180,E1 -2599.127,E2 -2599.127} C_VEL
LIN {X 0,Y 566.191,Z 752.35,A -85,B 0,C 180,E1 -2600.173,E2 -2600.173} C_VEL
LIN {X 0,Y 566.09,Z 761.63,A -85,B 0,C 180,E1 -2601.432,E2 -2601.432} C_VEL
LIN {X 0,Y 566.015,Z 768.138,A -85,B 0,C 180,E1 -2602.509,E2 -2602.509} C_VEL
LIN {X 0,Y 565.944,Z 773.521,A -85,B 0,C 180,E1 -2603.583,E2 -2603.583} C_VEL
LIN {X 0,Y 565.928,Z 777.926,A -85,B 0,C 180,E1 -2604.656,E2 -2604.656} C_VEL
LIN {X 0,Y 565.956,Z 781.448,A -85,B 0,C 180,E1 -2605.727,E2 -2605.727} C_VEL
LIN {X 0,Y 565.874,Z 784.802,A -85,B 0,C 180,E1 -2607.153,E2 -2607.153} C_VEL
LIN {X 0,Y 565.837,Z 786.008,A -85,B 0,C 180,E1 -2607.865,E2 -2607.865} C_VEL
LIN {X 0,Y 565.838,Z 787.297,A -85,B 0,C 180,E1 -2609.288,E2 -2609.288} C_VEL
LIN {X 0,Y 565.837,Z 787.5,A -85,B 0,C 180,E1 -2610,E2 -2610} C_VEL
LIN {X 0,Y 565.84,Z 786.811,A -85,B 0,C 180,E1 -2611.423,E2 -2611.423} C_VEL
LIN {X 0,Y 565.837,Z 786.008,A -85,B 0,C 180,E1 -2612.135,E2 -2612.135} C_VEL
LIN {X 0,Y 565.914,Z 783.322,A -85,B 0,C 180,E1 -2613.56,E2 -2613.56} C_VEL
LIN {X 0,Y 565.928,Z 780.395,A -85,B 0,C 180,E1 -2614.63,E2 -2614.63} C_VEL
LIN {X 0,Y 565.96,Z 775.093,A -85,B 0,C 180,E1 -2616.059,E2 -2616.059} C_VEL
LIN {X 0,Y 565.98,Z 770.038,A -85,B 0,C 180,E1 -2617.133,E2 -2617.133} C_VEL
LIN {X 0,Y 566.055,Z 763.892,A -85,B 0,C 180,E1 -2618.209,E2 -2618.209} C_VEL
LIN {X 0,Y 566.177,Z 756.532,A -85,B 0,C 180,E1 -2619.286,E2 -2619.286} C_VEL
LIN {X 0,Y 566.294,Z 747.72,A -85,B 0,C 180,E1 -2620.367,E2 -2620.367} C_VEL
LIN {X 0,Y 566.467,Z 736.006,A -85,B 0,C 180,E1 -2621.54,E2 -2621.54} C_VEL
LIN {X 0,Y 566.619,Z 724.889,A -85,B 0,C 180,E1 -2622.445,E2 -2622.445} C_VEL
LIN {X 0,Y 566.773,Z 714.187,A -85,B 0,C 180,E1 -2623.17,E2 -2623.17} C_VEL
LIN {X 0,Y 566.993,Z 702.812,A -85,B 0,C 180,E1 -2623.804,E2 -2623.804} C_VEL
LIN {X 0,Y 567.188,Z 689.429,A -85,B 0,C 180,E1 -2624.401,E2 -2624.401} C_VEL
LIN {X 0,Y 567.326,Z 675.216,A -85,B 0,C 180,E1 -2624.863,E2 -2624.863} C_VEL
LIN {X 0,Y 567.44,Z 662.688,A -85,B 0,C 180,E1 -2625.144,E2 -2625.144} C_VEL
LIN {X 0,Y 567.591,Z 619.868,A -85,B 0,C 180,E1 -2625.715,E2 -2625.715} C_VEL
LIN {X 0,Y 567.667,Z 532.087,A -85,B 0,C 180,E1 -2626.846,E2 -2626.846} C_VEL
LIN {X 0,Y 566.563,Z 526.192,A -85,B 0,C 180,E1 -2626.975,E2 -2626.975} C_VEL
LIN {X 0,Y 566.577,Z 519.08,A -85,B 0,C 180,E1 -2628.065,E2 -2628.065} C_VEL
LIN {X 0,Y 566.849,Z 500.473,A -85,B 0,C 180,E1 -2631.072,E2 -2631.072} C_VEL
LIN {X 0,Y 567.095,Z 484.157,A -85,B 0,C 180,E1 -2633.757,E2 -2633.757} C_VEL
LIN {X 0,Y 567.171,Z 474.17,A -85,B 0,C 180,E1 -2635.416,E2 -2635.416} C_VEL
LIN {X 0,Y 566.218,Z 469.156,A -85,B 0,C 180,E1 -2636.342,E2 -2636.342} C_VEL
